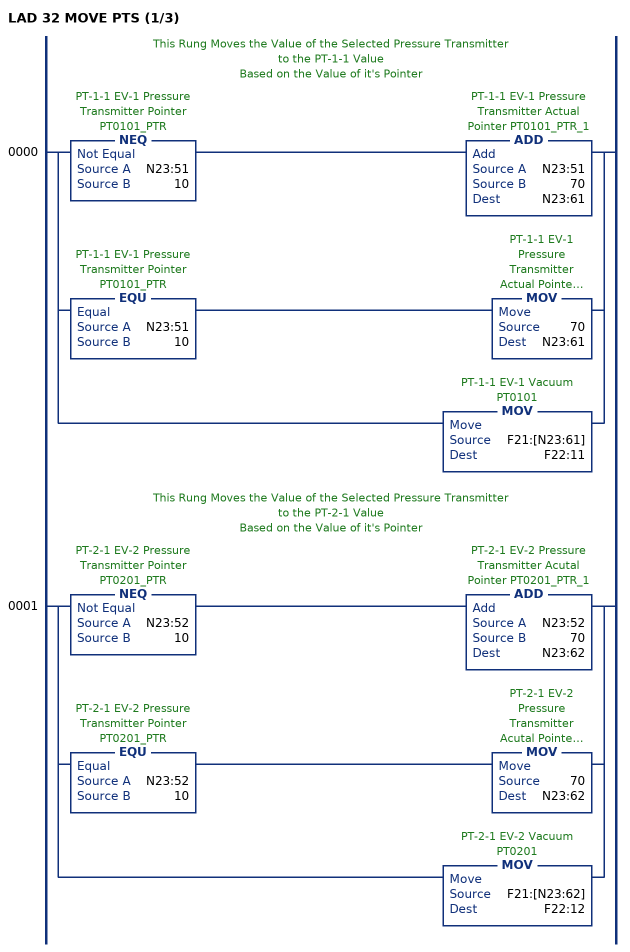
% Rung: 0 %
% This Rung Moves the Value of the Selected Pressure Transmitter
% to the PT-1-1 Value
% Based on the Value of it's Pointer %
SOR BST NEQ N23:51 10 ADD N23:51 70 N23:61 NXB EQU N23:51 10 MOV 70 N23:61 NXB MOV F21:[N23:61] F22:11 BND EOR
%   N23:51  PT0101_PTR  "PT-1-1 EV-1 Pressure Transmitter Pointer" %
%   N23:61  PT0101_PTR_1  "PT-1-1 EV-1 Pressure Transmitter Actual Pointer" %
%   F22:11  PT0101  "PT-1-1 EV-1 Vacuum" %
% Rung: 1 %
% This Rung Moves the Value of the Selected Pressure Transmitter
% to the PT-2-1 Value
% Based on the Value of it's Pointer %
SOR BST NEQ N23:52 10 ADD N23:52 70 N23:62 NXB EQU N23:52 10 MOV 70 N23:62 NXB MOV F21:[N23:62] F22:12 BND EOR
%   N23:52  PT0201_PTR  "PT-2-1 EV-2 Pressure Transmitter Pointer" %
%   N23:62  PT0201_PTR_1  "PT-2-1 EV-2 Pressure Transmitter Acutal Pointer" %
%   F22:12  PT0201  "PT-2-1 EV-2 Vacuum" %

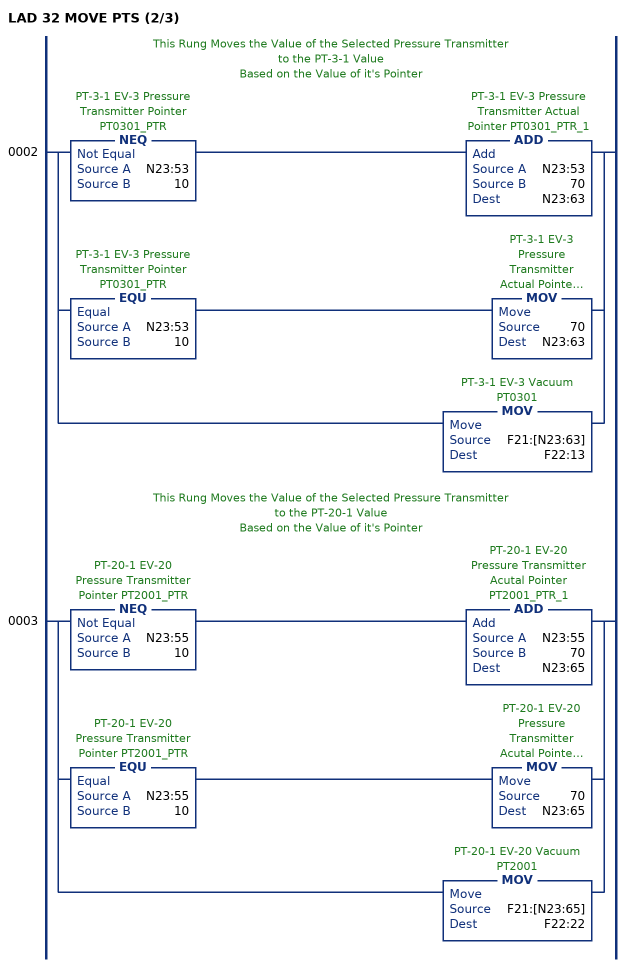
% Rung: 2 %
% This Rung Moves the Value of the Selected Pressure Transmitter
% to the PT-3-1 Value
% Based on the Value of it's Pointer %
SOR BST NEQ N23:53 10 ADD N23:53 70 N23:63 NXB EQU N23:53 10 MOV 70 N23:63 NXB MOV F21:[N23:63] F22:13 BND EOR
%   N23:53  PT0301_PTR  "PT-3-1 EV-3 Pressure Transmitter Pointer" %
%   N23:63  PT0301_PTR_1  "PT-3-1 EV-3 Pressure Transmitter Actual Pointer" %
%   F22:13  PT0301  "PT-3-1 EV-3 Vacuum" %
% Rung: 3 %
% This Rung Moves the Value of the Selected Pressure Transmitter
% to the PT-20-1 Value
% Based on the Value of it's Pointer %
SOR BST NEQ N23:55 10 ADD N23:55 70 N23:65 NXB EQU N23:55 10 MOV 70 N23:65 NXB MOV F21:[N23:65] F22:22 BND EOR
%   N23:55  PT2001_PTR  "PT-20-1 EV-20 Pressure Transmitter Pointer" %
%   N23:65  PT2001_PTR_1  "PT-20-1 EV-20 Pressure Transmitter Acutal Pointer" %
%   F22:22  PT2001  "PT-20-1 EV-20 Vacuum" %

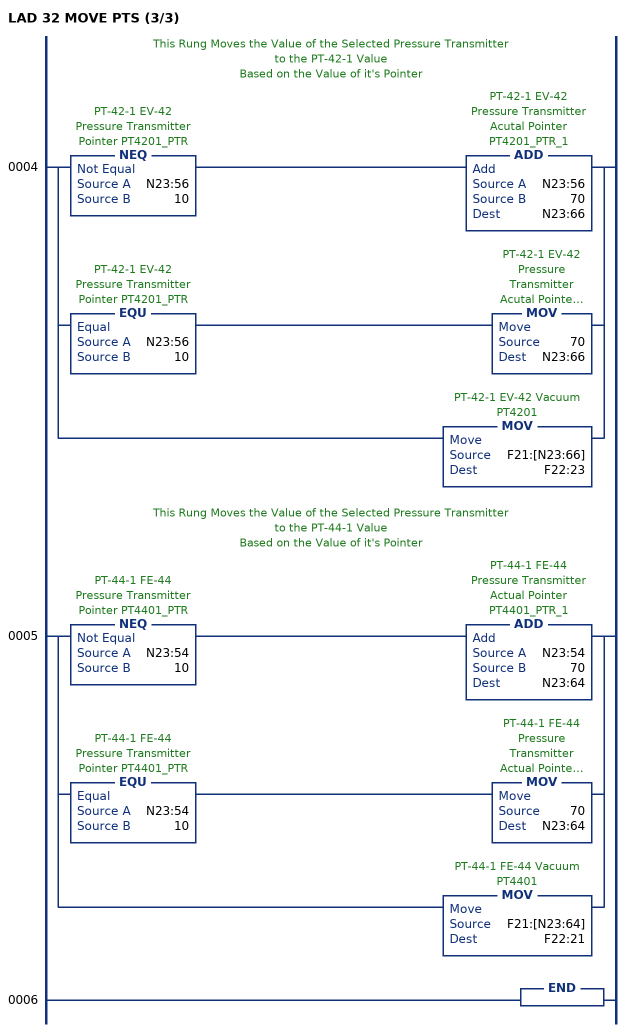
% Rung: 4 %
% This Rung Moves the Value of the Selected Pressure Transmitter
% to the PT-42-1 Value
% Based on the Value of it's Pointer %
SOR BST NEQ N23:56 10 ADD N23:56 70 N23:66 NXB EQU N23:56 10 MOV 70 N23:66 NXB MOV F21:[N23:66] F22:23 BND EOR
%   N23:56  PT4201_PTR  "PT-42-1 EV-42 Pressure Transmitter Pointer" %
%   N23:66  PT4201_PTR_1  "PT-42-1 EV-42 Pressure Transmitter Acutal Pointer" %
%   F22:23  PT4201  "PT-42-1 EV-42 Vacuum" %
% Rung: 5 %
% This Rung Moves the Value of the Selected Pressure Transmitter
% to the PT-44-1 Value
% Based on the Value of it's Pointer %
SOR BST NEQ N23:54 10 ADD N23:54 70 N23:64 NXB EQU N23:54 10 MOV 70 N23:64 NXB MOV F21:[N23:64] F22:21 BND EOR
%   N23:54  PT4401_PTR  "PT-44-1 FE-44 Pressure Transmitter Pointer" %
%   N23:64  PT4401_PTR_1  "PT-44-1 FE-44 Pressure Transmitter Actual Pointer" %
%   F22:21  PT4401  "PT-44-1 FE-44 Vacuum" %
% Rung: 6 %
SOR END EOR

LADDER 33 "MOVE FTS"    % Move FT Info to Sequencial Locations, etc %
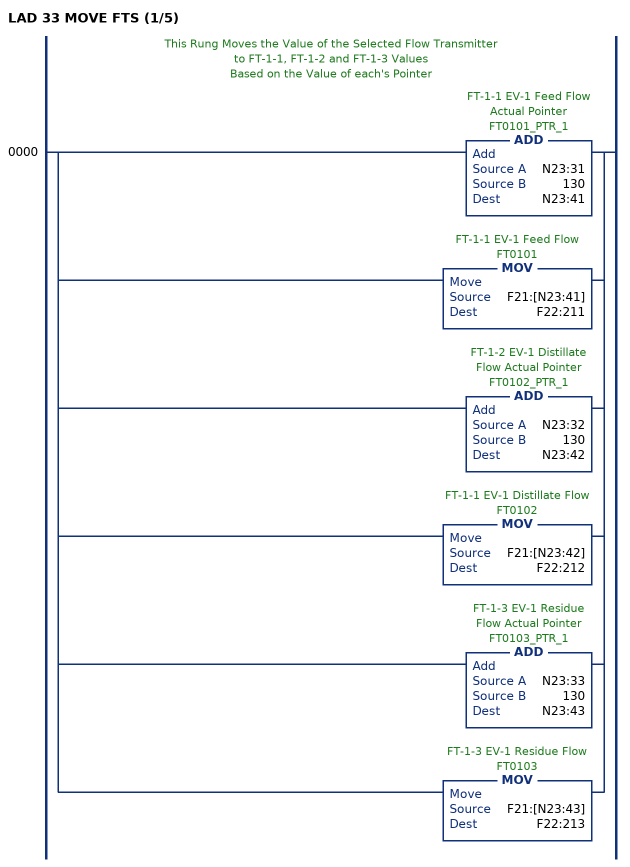
% Rung: 0 %
% This Rung Moves the Value of the Selected Flow Transmitter
% to FT-1-1, FT-1-2 and FT-1-3 Values
% Based on the Value of each's Pointer %
SOR BST ADD N23:31 130 N23:41 NXB MOV F21:[N23:41] F22:211 NXB ADD N23:32 130 N23:42 NXB MOV F21:[N23:42] F22:212 NXB ADD N23:33 130 N23:43 NXB MOV F21:[N23:43] F22:213 BND EOR
%   N23:31  FT0101_PTR  "FT-1-1 EV-1 Feed Flow Pointer" %
%   N23:41  FT0101_PTR_1  "FT-1-1 EV-1 Feed Flow Actual Pointer" %
%   F22:211  FT0101  "FT-1-1 EV-1 Feed Flow" %
%   N23:32  FT0102_PTR  "FT-1-2 EV-1 Distillate Flow Pointer" %
%   N23:42  FT0102_PTR_1  "FT-1-2 EV-1 Distillate Flow Actual Pointer" %
%   F22:212  FT0102  "FT-1-1 EV-1 Distillate Flow" %
%   N23:33  FT0103_PTR  "FT-1-3 EV-1 Residue Flow Pointer" %
%   N23:43  FT0103_PTR_1  "FT-1-3 EV-1 Residue Flow Actual Pointer" %
%   F22:213  FT0103  "FT-1-3 EV-1 Residue Flow" %

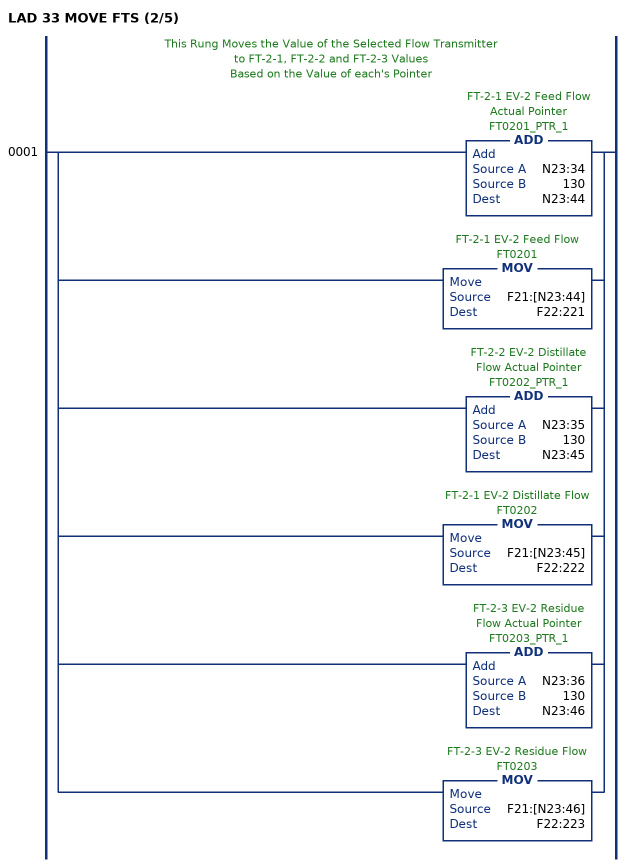
% Rung: 1 %
% This Rung Moves the Value of the Selected Flow Transmitter
% to FT-2-1, FT-2-2 and FT-2-3 Values
% Based on the Value of each's Pointer %
SOR BST ADD N23:34 130 N23:44 NXB MOV F21:[N23:44] F22:221 NXB ADD N23:35 130 N23:45 NXB MOV F21:[N23:45] F22:222 NXB ADD N23:36 130 N23:46 NXB MOV F21:[N23:46] F22:223 BND EOR
%   N23:34  FT0201_PTR  "FT-2-1 EV-2 Feed Flow Pointer" %
%   N23:44  FT0201_PTR_1  "FT-2-1 EV-2 Feed Flow Actual Pointer" %
%   F22:221  FT0201  "FT-2-1 EV-2 Feed Flow" %
%   N23:35  FT0202_PTR  "FT-2-2 EV-2 Distillate Flow Pointer" %
%   N23:45  FT0202_PTR_1  "FT-2-2 EV-2 Distillate Flow Actual Pointer" %
%   F22:222  FT0202  "FT-2-1 EV-2 Distillate Flow" %
%   N23:36  FT0203_PTR  "FT-2-3 EV-2 Residue Flow Pointer" %
%   N23:46  FT0203_PTR_1  "FT-2-3 EV-2 Residue Flow Actual Pointer" %
%   F22:223  FT0203  "FT-2-3 EV-2 Residue Flow" %

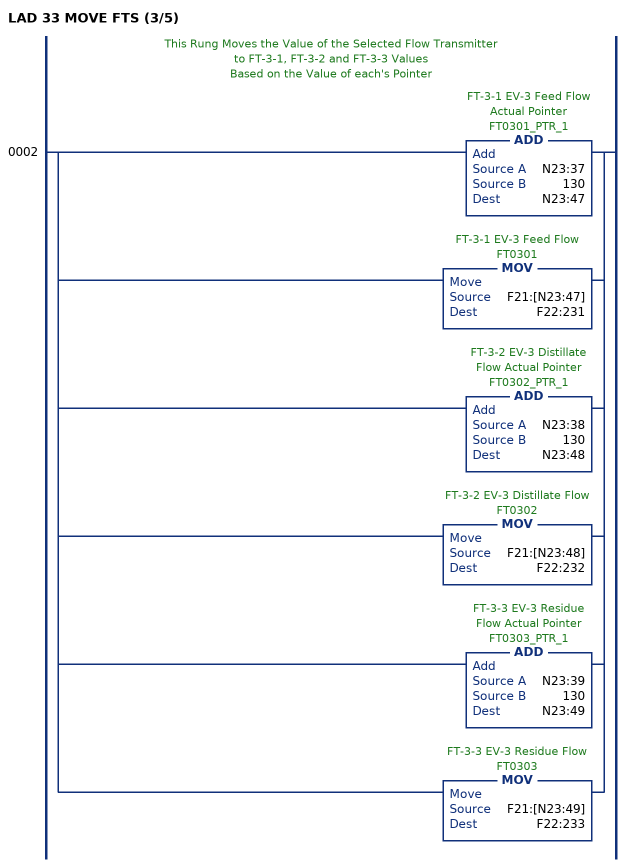
% Rung: 2 %
% This Rung Moves the Value of the Selected Flow Transmitter
% to FT-3-1, FT-3-2 and FT-3-3 Values
% Based on the Value of each's Pointer %
SOR BST ADD N23:37 130 N23:47 NXB MOV F21:[N23:47] F22:231 NXB ADD N23:38 130 N23:48 NXB MOV F21:[N23:48] F22:232 NXB ADD N23:39 130 N23:49 NXB MOV F21:[N23:49] F22:233 BND EOR
%   N23:37  FT0301_PTR  "FT-3-1 EV-3 Feed Flow Pointer" %
%   N23:47  FT0301_PTR_1  "FT-3-1 EV-3 Feed Flow Actual Pointer" %
%   F22:231  FT0301  "FT-3-1 EV-3 Feed Flow" %
%   N23:38  FT0302_PTR  "FT-3-2 EV-3 Distillate Flow Pointer" %
%   N23:48  FT0302_PTR_1  "FT-3-2 EV-3 Distillate Flow Actual Pointer" %
%   F22:232  FT0302  "FT-3-2 EV-3 Distillate Flow" %
%   N23:39  FT0303_PTR  "FT-3-3 EV-3 Residue Flow Pointer" %
%   N23:49  FT0303_PTR_1  "FT-3-3 EV-3 Residue Flow Actual Pointer" %
%   F22:233  FT0303  "FT-3-3 EV-3 Residue Flow" %

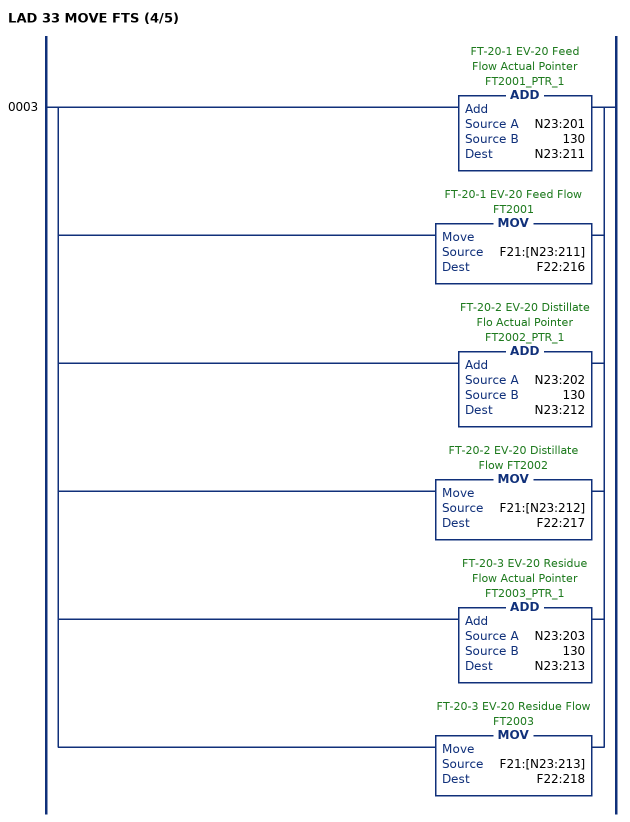
% Rung: 3 %
SOR BST ADD N23:201 130 N23:211 NXB MOV F21:[N23:211] F22:216 NXB ADD N23:202 130 N23:212 NXB MOV F21:[N23:212] F22:217 NXB ADD N23:203 130 N23:213 NXB MOV F21:[N23:213] F22:218 BND EOR
%   N23:201  FT2001_PTR  "FT-20-1 EV-20 Feed Flow Pointer" %
%   N23:211  FT2001_PTR_1  "FT-20-1 EV-20 Feed Flow Actual Pointer" %
%   F22:216  FT2001  "FT-20-1 EV-20 Feed Flow" %
%   N23:202  FT2002_PTR  "FT-20-2 EV-20 Distillate Flo Pointer" %
%   N23:212  FT2002_PTR_1  "FT-20-2 EV-20 Distillate Flo Actual Pointer" %
%   F22:217  FT2002  "FT-20-2 EV-20 Distillate Flow" %
%   N23:203  FT2003_PTR  "FT-20-3 EV-20 Residue Flow Pointer" %
%   N23:213  FT2003_PTR_1  "FT-20-3 EV-20 Residue Flow Actual Pointer" %
%   F22:218  FT2003  "FT-20-3 EV-20 Residue Flow" %

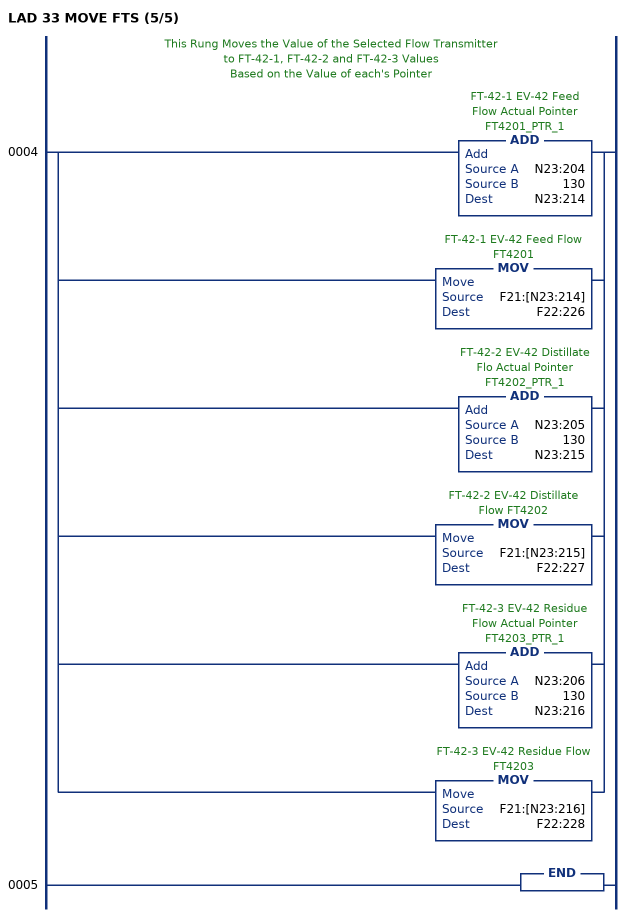
% Rung: 4 %
% This Rung Moves the Value of the Selected Flow Transmitter
% to FT-42-1, FT-42-2 and FT-42-3 Values
% Based on the Value of each's Pointer %
SOR BST ADD N23:204 130 N23:214 NXB MOV F21:[N23:214] F22:226 NXB ADD N23:205 130 N23:215 NXB MOV F21:[N23:215] F22:227 NXB ADD N23:206 130 N23:216 NXB MOV F21:[N23:216] F22:228 BND EOR
%   N23:204  FT4201_PTR  "FT-42-1 EV-42 Feed Flow Pointer" %
%   N23:214  FT4201_PTR_1  "FT-42-1 EV-42 Feed Flow Actual Pointer" %
%   F22:226  FT4201  "FT-42-1 EV-42 Feed Flow" %
%   N23:205  FT4202_PTR  "FT-42-2 EV-42 Distillate Flo Pointer" %
%   N23:215  FT4202_PTR_1  "FT-42-2 EV-42 Distillate Flo Actual Pointer" %
%   F22:227  FT4202  "FT-42-2 EV-42 Distillate Flow" %
%   N23:206  FT4203_PTR  "FT-42-3 EV-42 Residue Flow Pointer" %
%   N23:216  FT4203_PTR_1  "FT-42-3 EV-42 Residue Flow Actual Pointer" %
%   F22:228  FT4203  "FT-42-3 EV-42 Residue Flow" %
% Rung: 5 %
SOR END EOR

LADDER 34 "CALC WTS"    % Convert Remote I/O Data to Real Data for All Scale %
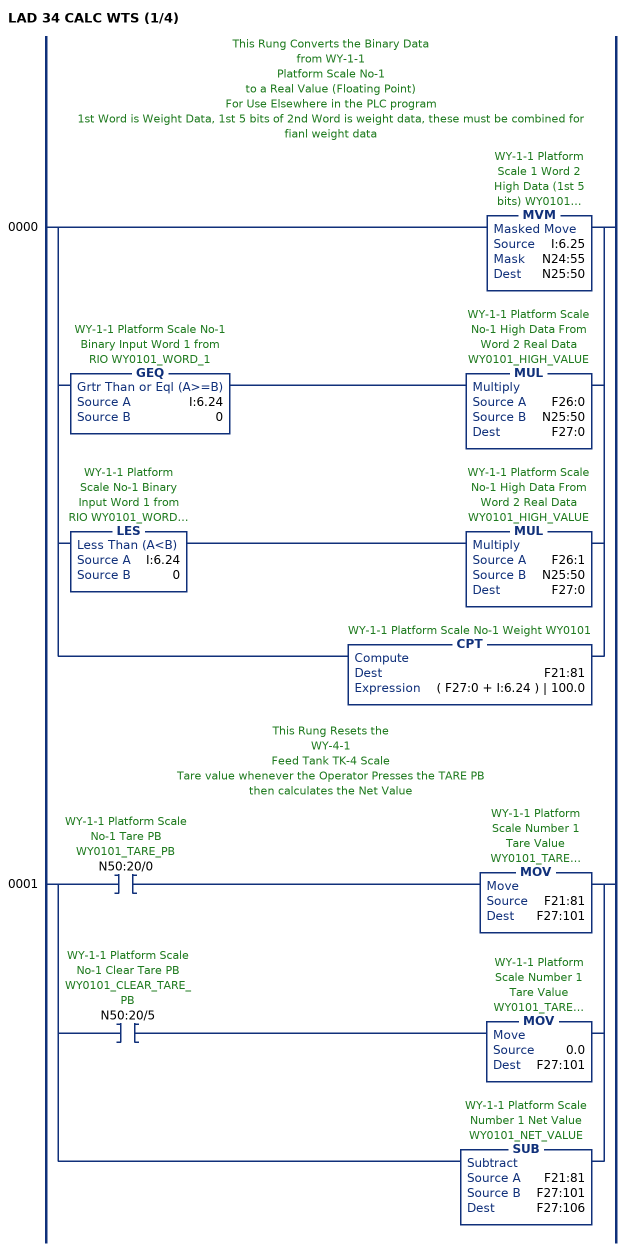
% Rung: 0 %
% This Rung Converts the Binary Data
% from WY-1-1
% Platform Scale No-1
% to a Real Value (Floating Point)
% For Use Elsewhere in the PLC program
% 1st Word is Weight Data, 1st 5 bits of 2nd Word is weight data, these must be combined for fianl weight data %
SOR BST MVM I:6.25 N24:55 N25:50 NXB GEQ I:6.24 0 MUL F26:0 N25:50 F27:0 NXB LES I:6.24 0 MUL F26:1 N25:50 F27:0 NXB CPT F21:81 " ( F27:0 + I:6.24 ) | 100.0 " BND EOR
%   I:6.25  WY0101_WORD_2  "WY-1-1 Platform Scale No-1 Binary Input Word 2 from RIO" %
%   N24:55  WY0101_MASK  "WY-1-1 Platform Scale No-1 Word 2 Mask (Use 1st 5 bits)" %
%   N25:50  WY0101_HIGH_DATA  "WY-1-1 Platform Scale 1 Word 2 High Data (1st 5 bits)" %
%   I:6.24  WY0101_WORD_1  "WY-1-1 Platform Scale No-1 Binary Input Word 1 from RIO" %
%   F26:0  WT_MULTIPLIER_1  "Weigh Scale Multipler if Word 1 >= 0" %
%   F27:0  WY0101_HIGH_VALUE  "WY-1-1 Platform Scale No-1 High Data From Word 2 Real Data" %
%   F26:1  WT_MULTIPLIER_2  "Weigh Scale Multipler if Word 1 < 0" %
%   F21:81  WY0101  "WY-1-1 Platform Scale No-1 Weight" %
% Rung: 1 %
% This Rung Resets the
% WY-4-1
% Feed Tank TK-4 Scale
% Tare value whenever the Operator Presses the TARE PB
% then calculates the Net Value %
SOR BST XIC N50:20/0 MOV F21:81 F27:101 NXB XIC N50:20/5 MOV 0.0 F27:101 NXB SUB F21:81 F27:101 F27:106 BND EOR
%   N50:20/0  WY0101_TARE_PB  "WY-1-1 Platform Scale No-1 Tare PB" %
%   F21:81  WY0101  "WY-1-1 Platform Scale No-1 Weight" %
%   F27:101  WY0101_TARE_VALUE  "WY-1-1 Platform Scale Number 1 Tare Value" %
%   N50:20/5  WY0101_CLEAR_TARE_PB  "WY-1-1 Platform Scale No-1 Clear Tare PB" %
%   F27:106  WY0101_NET_VALUE  "WY-1-1 Platform Scale Number 1 Net Value" %

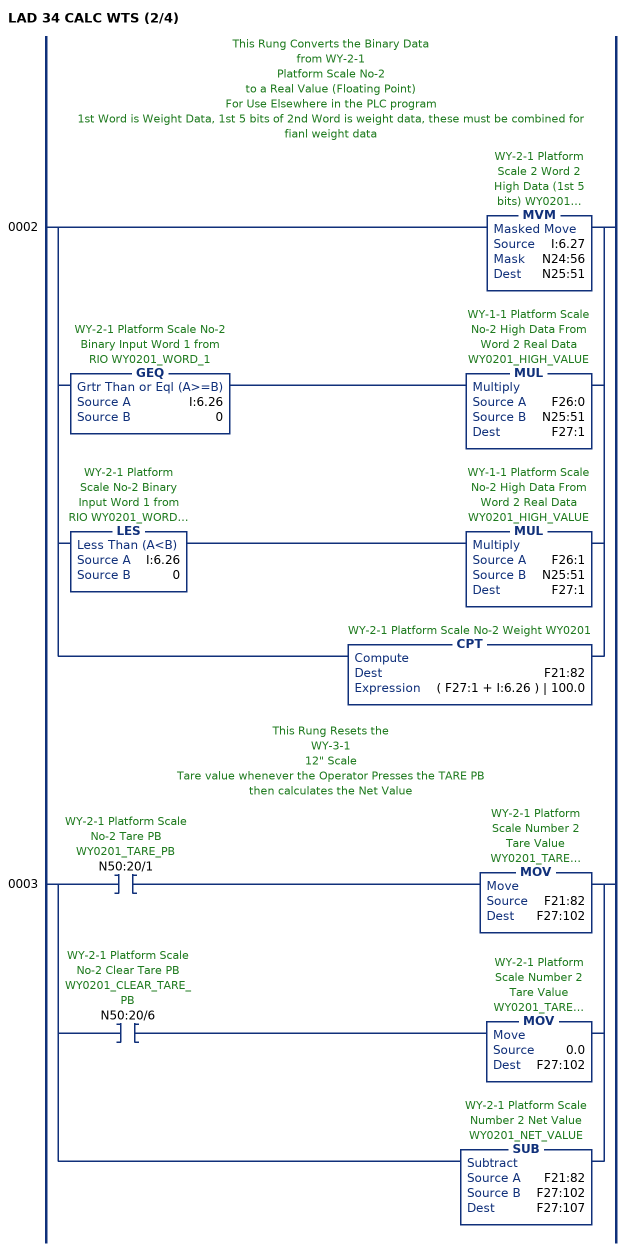
% Rung: 2 %
% This Rung Converts the Binary Data
% from WY-2-1
% Platform Scale No-2
% to a Real Value (Floating Point)
% For Use Elsewhere in the PLC program
% 1st Word is Weight Data, 1st 5 bits of 2nd Word is weight data, these must be combined for fianl weight data %
SOR BST MVM I:6.27 N24:56 N25:51 NXB GEQ I:6.26 0 MUL F26:0 N25:51 F27:1 NXB LES I:6.26 0 MUL F26:1 N25:51 F27:1 NXB CPT F21:82 " ( F27:1 + I:6.26 ) | 100.0 " BND EOR
%   I:6.27  WY0201_WORD_2  "WY-2-1 Platform Scale No-2 Binary Input Word 2 from RIO" %
%   N24:56  WY0201_MASK  "WY-2-1 Platform Scale No-2 Word 2 Mask (Use 1st 5 bits)" %
%   N25:51  WY0201_HIGH_DATA  "WY-2-1 Platform Scale 2 Word 2 High Data (1st 5 bits)" %
%   I:6.26  WY0201_WORD_1  "WY-2-1 Platform Scale No-2 Binary Input Word 1 from RIO" %
%   F26:0  WT_MULTIPLIER_1  "Weigh Scale Multipler if Word 1 >= 0" %
%   F27:1  WY0201_HIGH_VALUE  "WY-1-1 Platform Scale No-2 High Data From Word 2 Real Data" %
%   F26:1  WT_MULTIPLIER_2  "Weigh Scale Multipler if Word 1 < 0" %
%   F21:82  WY0201  "WY-2-1 Platform Scale No-2 Weight" %
% Rung: 3 %
% This Rung Resets the
% WY-3-1
% 12" Scale
% Tare value whenever the Operator Presses the TARE PB
% then calculates the Net Value %
SOR BST XIC N50:20/1 MOV F21:82 F27:102 NXB XIC N50:20/6 MOV 0.0 F27:102 NXB SUB F21:82 F27:102 F27:107 BND EOR
%   N50:20/1  WY0201_TARE_PB  "WY-2-1 Platform Scale No-2 Tare PB" %
%   F21:82  WY0201  "WY-2-1 Platform Scale No-2 Weight" %
%   F27:102  WY0201_TARE_VALUE  "WY-2-1 Platform Scale Number 2 Tare Value" %
%   N50:20/6  WY0201_CLEAR_TARE_PB  "WY-2-1 Platform Scale No-2 Clear Tare PB" %
%   F27:107  WY0201_NET_VALUE  "WY-2-1 Platform Scale Number 2 Net Value" %

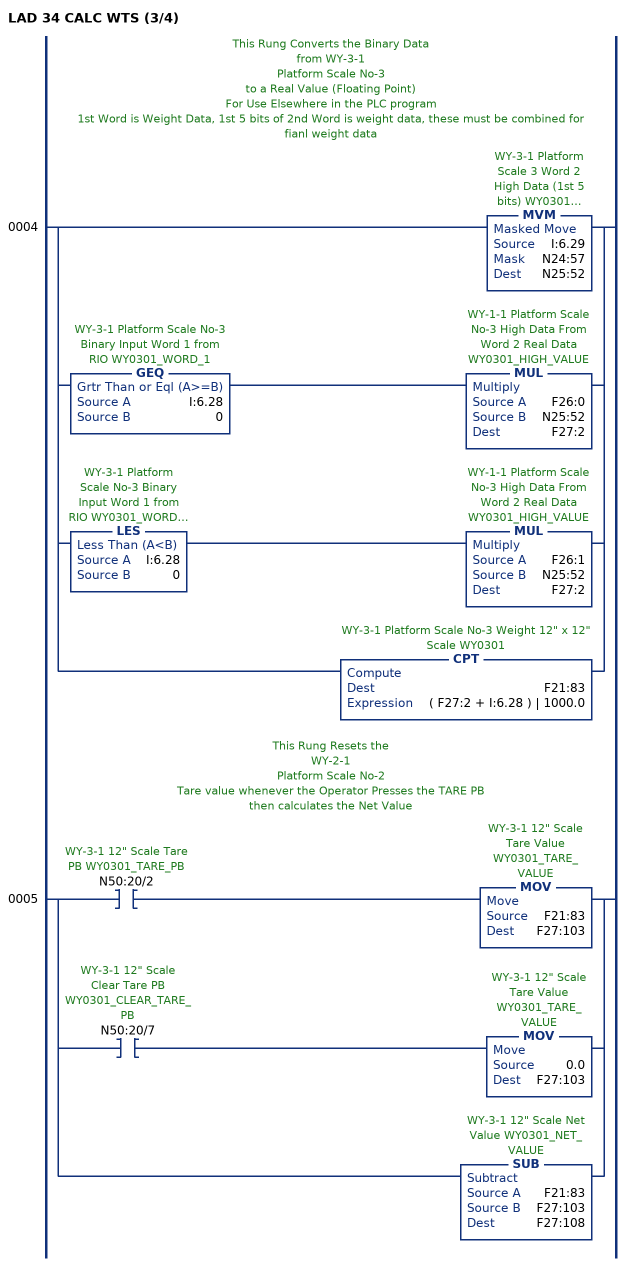
% Rung: 4 %
% This Rung Converts the Binary Data
% from WY-3-1
% Platform Scale No-3
% to a Real Value (Floating Point)
% For Use Elsewhere in the PLC program
% 1st Word is Weight Data, 1st 5 bits of 2nd Word is weight data, these must be combined for fianl weight data %
SOR BST MVM I:6.29 N24:57 N25:52 NXB GEQ I:6.28 0 MUL F26:0 N25:52 F27:2 NXB LES I:6.28 0 MUL F26:1 N25:52 F27:2 NXB CPT F21:83 " ( F27:2 + I:6.28 ) | 1000.0 " BND EOR
%   I:6.29  WY0301_WORD_2  "WY-3-1 Platform Scale No-3 Binary Input Word 2 from RIO" %
%   N24:57  WY0301_MASK  "WY-3-1 Platform Scale No-3 Word 2 Mask (Use 1st 5 bits)" %
%   N25:52  WY0301_HIGH_DATA  "WY-3-1 Platform Scale 3 Word 2 High Data (1st 5 bits)" %
%   I:6.28  WY0301_WORD_1  "WY-3-1 Platform Scale No-3 Binary Input Word 1 from RIO" %
%   F26:0  WT_MULTIPLIER_1  "Weigh Scale Multipler if Word 1 >= 0" %
%   F27:2  WY0301_HIGH_VALUE  "WY-1-1 Platform Scale No-3 High Data From Word 2 Real Data" %
%   F26:1  WT_MULTIPLIER_2  "Weigh Scale Multipler if Word 1 < 0" %
%   F21:83  WY0301  "WY-3-1 Platform Scale No-3 Weight 12" x 12" Scale" %
% Rung: 5 %
% This Rung Resets the
% WY-2-1
% Platform Scale No-2
% Tare value whenever the Operator Presses the TARE PB
% then calculates the Net Value %
SOR BST XIC N50:20/2 MOV F21:83 F27:103 NXB XIC N50:20/7 MOV 0.0 F27:103 NXB SUB F21:83 F27:103 F27:108 BND EOR
%   N50:20/2  WY0301_TARE_PB  "WY-3-1 12" Scale Tare PB" %
%   F21:83  WY0301  "WY-3-1 Platform Scale No-3 Weight 12" x 12" Scale" %
%   F27:103  WY0301_TARE_VALUE  "WY-3-1 12" Scale Tare Value" %
%   N50:20/7  WY0301_CLEAR_TARE_PB  "WY-3-1 12" Scale Clear Tare PB" %
%   F27:108  WY0301_NET_VALUE  "WY-3-1 12" Scale Net Value" %

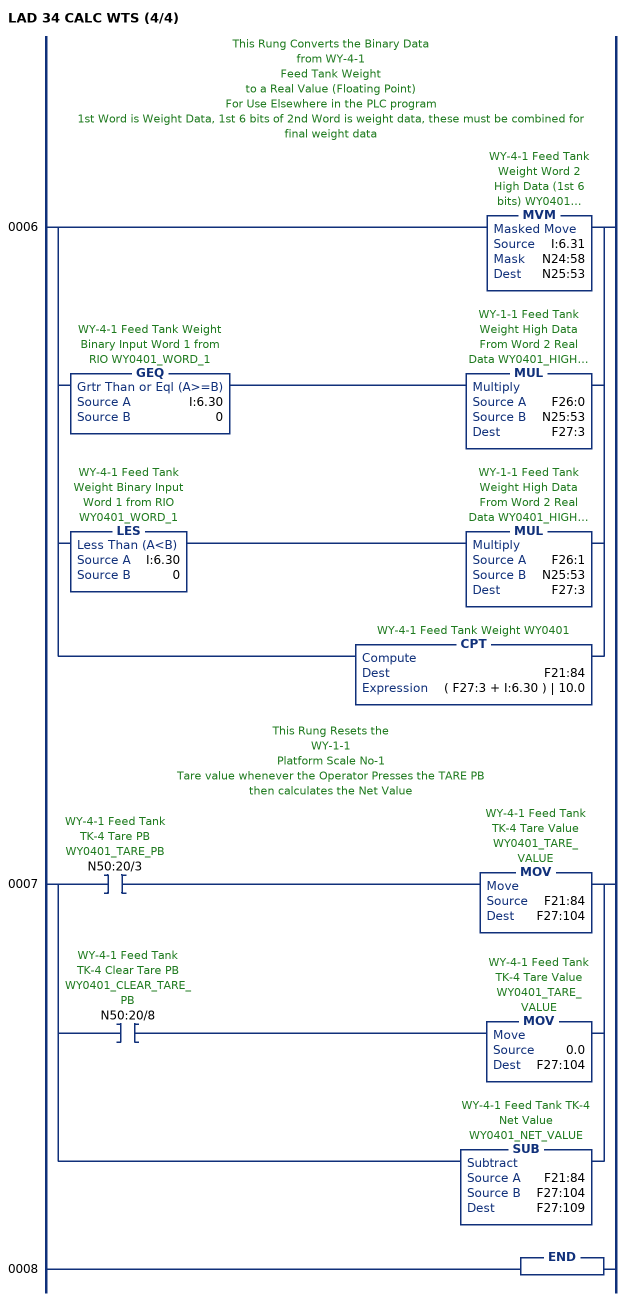
% Rung: 6 %
% This Rung Converts the Binary Data
% from WY-4-1
% Feed Tank Weight
% to a Real Value (Floating Point)
% For Use Elsewhere in the PLC program
% 1st Word is Weight Data, 1st 6 bits of 2nd Word is weight data, these must be combined for final weight data %
SOR BST MVM I:6.31 N24:58 N25:53 NXB GEQ I:6.30 0 MUL F26:0 N25:53 F27:3 NXB LES I:6.30 0 MUL F26:1 N25:53 F27:3 NXB CPT F21:84 " ( F27:3 + I:6.30 ) | 10.0 " BND EOR
%   I:6.31  WY0401_WORD_2  "WY-4-1 Feed Tank Weight Binary Input Word 2 from RIO" %
%   N24:58  WY0401_MASK  "WY-4-1 Feed Tank Weight Word 2 Mask (Use 1st 6 bits)" %
%   N25:53  WY0401_HIGH_DATA  "WY-4-1 Feed Tank Weight Word 2 High Data (1st 6 bits)" %
%   I:6.30  WY0401_WORD_1  "WY-4-1 Feed Tank Weight Binary Input Word 1 from RIO" %
%   F26:0  WT_MULTIPLIER_1  "Weigh Scale Multipler if Word 1 >= 0" %
%   F27:3  WY0401_HIGH_VALUE  "WY-1-1 Feed Tank Weight High Data From Word 2 Real Data" %
%   F26:1  WT_MULTIPLIER_2  "Weigh Scale Multipler if Word 1 < 0" %
%   F21:84  WY0401  "WY-4-1 Feed Tank Weight" %
% Rung: 7 %
% This Rung Resets the
% WY-1-1
% Platform Scale No-1
% Tare value whenever the Operator Presses the TARE PB
% then calculates the Net Value %
SOR BST XIC N50:20/3 MOV F21:84 F27:104 NXB XIC N50:20/8 MOV 0.0 F27:104 NXB SUB F21:84 F27:104 F27:109 BND EOR
%   N50:20/3  WY0401_TARE_PB  "WY-4-1 Feed Tank TK-4 Tare PB" %
%   F21:84  WY0401  "WY-4-1 Feed Tank Weight" %
%   F27:104  WY0401_TARE_VALUE  "WY-4-1 Feed Tank TK-4 Tare Value" %
%   N50:20/8  WY0401_CLEAR_TARE_PB  "WY-4-1 Feed Tank TK-4 Clear Tare PB" %
%   F27:109  WY0401_NET_VALUE  "WY-4-1 Feed Tank TK-4 Net Value" %
% Rung: 8 %
SOR END EOR

LADDER 35 "CALC WT FT"    % Calcualte Flow Rates based on Weight Changes %
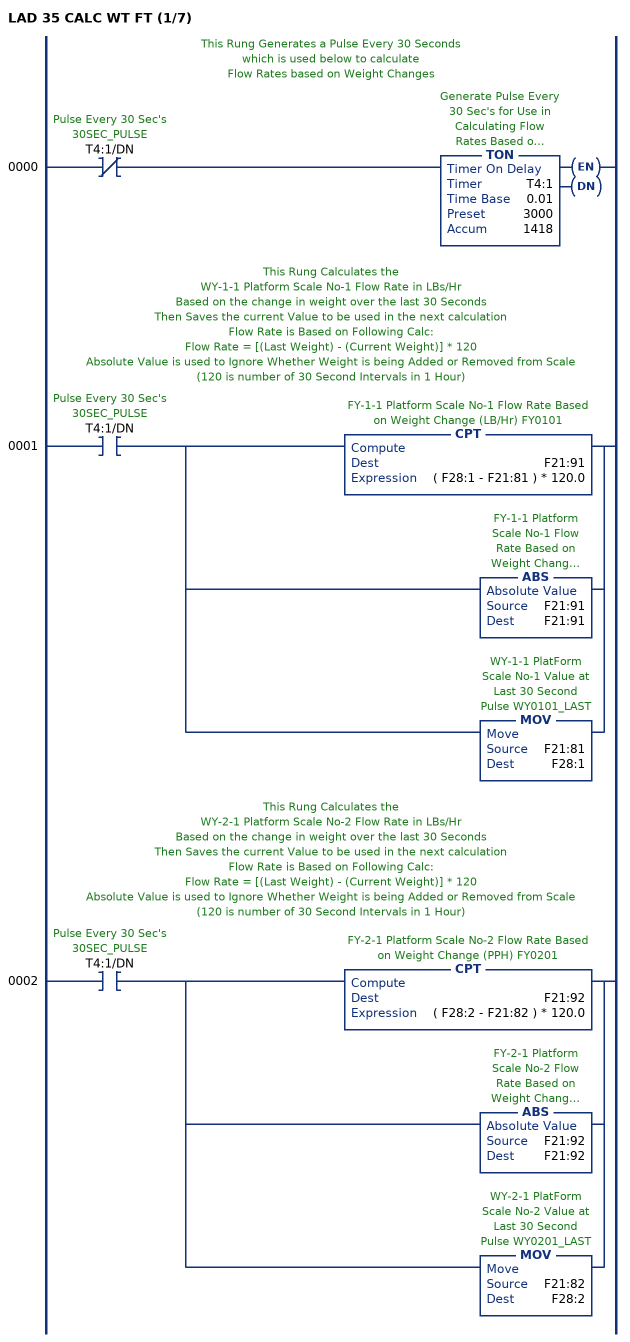
% Rung: 0 %
% This Rung Generates a Pulse Every 30 Seconds
% which is used below to calculate
% Flow Rates based on Weight Changes %
SOR XIO T4:1/DN TON T4:1 0.01 3000 1418 EOR
%   T4:1/DN  30SEC_PULSE  "Pulse Every 30 Sec's" %
%   T4:1  30SEC_TIMER  "Generate Pulse Every 30 Sec's for Use in Calculating Flow Rates Based on Weigh" %
% Rung: 1 %
% This Rung Calculates the
% WY-1-1 Platform Scale No-1 Flow Rate in LBs/Hr
% Based on the change in weight over the last 30 Seconds
% Then Saves the current Value to be used in the next calculation
% Flow Rate is Based on Following Calc:
% 
% Flow Rate = [(Last Weight) - (Current Weight)] * 120
% 
% Absolute Value is used to Ignore Whether Weight is being Added or Removed from Scale
% (120 is number of 30 Second Intervals in 1 Hour) %
SOR XIC T4:1/DN BST CPT F21:91 " ( F28:1 - F21:81 ) * 120.0 " NXB ABS F21:91 F21:91 NXB MOV F21:81 F28:1 BND EOR
%   T4:1/DN  30SEC_PULSE  "Pulse Every 30 Sec's" %
%   F21:91  FY0101  "FY-1-1 Platform Scale No-1 Flow Rate Based on Weight Change (LB/Hr)" %
%   F28:1  WY0101_LAST  "WY-1-1 PlatForm Scale No-1 Value at Last 30 Second Pulse" %
%   F21:81  WY0101  "WY-1-1 Platform Scale No-1 Weight" %
% Rung: 2 %
% This Rung Calculates the
% WY-2-1 Platform Scale No-2 Flow Rate in LBs/Hr
% Based on the change in weight over the last 30 Seconds
% Then Saves the current Value to be used in the next calculation
% Flow Rate is Based on Following Calc:
% 
% Flow Rate = [(Last Weight) - (Current Weight)] * 120
% 
% Absolute Value is used to Ignore Whether Weight is being Added or Removed from Scale
% (120 is number of 30 Second Intervals in 1 Hour) %
SOR XIC T4:1/DN BST CPT F21:92 " ( F28:2 - F21:82 ) * 120.0 " NXB ABS F21:92 F21:92 NXB MOV F21:82 F28:2 BND EOR
%   T4:1/DN  30SEC_PULSE  "Pulse Every 30 Sec's" %
%   F21:92  FY0201  "FY-2-1 Platform Scale No-2 Flow Rate Based on Weight Change (PPH)" %
%   F28:2  WY0201_LAST  "WY-2-1 PlatForm Scale No-2 Value at Last 30 Second Pulse" %
%   F21:82  WY0201  "WY-2-1 Platform Scale No-2 Weight" %

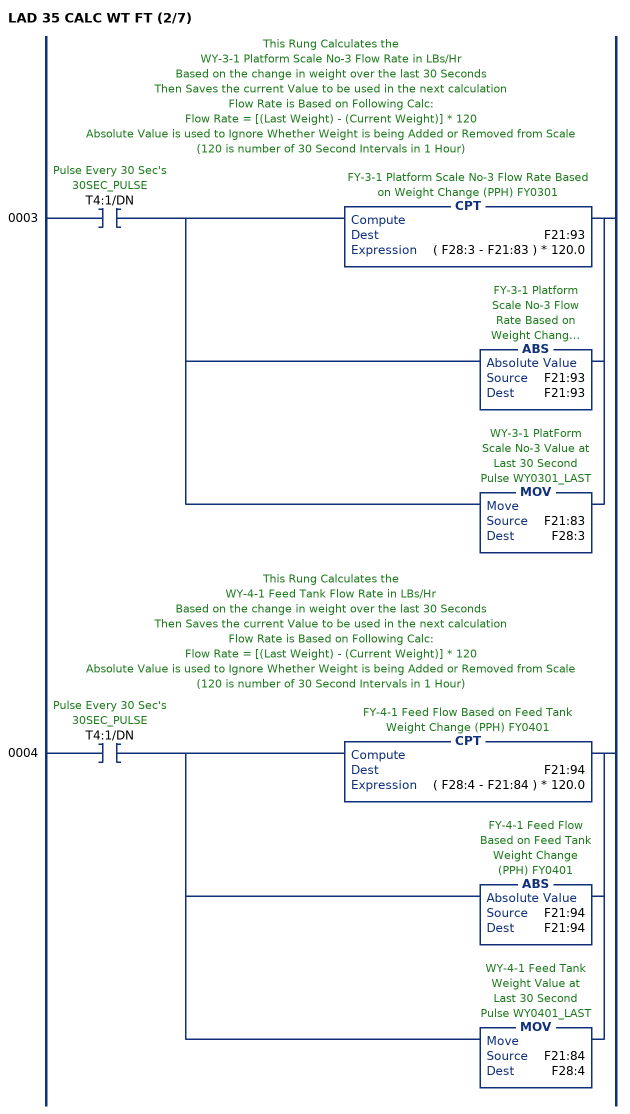
% Rung: 3 %
% This Rung Calculates the
% WY-3-1 Platform Scale No-3 Flow Rate in LBs/Hr
% Based on the change in weight over the last 30 Seconds
% Then Saves the current Value to be used in the next calculation
% Flow Rate is Based on Following Calc:
% 
% Flow Rate = [(Last Weight) - (Current Weight)] * 120
% 
% Absolute Value is used to Ignore Whether Weight is being Added or Removed from Scale
% (120 is number of 30 Second Intervals in 1 Hour) %
SOR XIC T4:1/DN BST CPT F21:93 " ( F28:3 - F21:83 ) * 120.0 " NXB ABS F21:93 F21:93 NXB MOV F21:83 F28:3 BND EOR
%   T4:1/DN  30SEC_PULSE  "Pulse Every 30 Sec's" %
%   F21:93  FY0301  "FY-3-1 Platform Scale No-3 Flow Rate Based on Weight Change (PPH)" %
%   F28:3  WY0301_LAST  "WY-3-1 PlatForm Scale No-3 Value at Last 30 Second Pulse" %
%   F21:83  WY0301  "WY-3-1 Platform Scale No-3 Weight 12" x 12" Scale" %
% Rung: 4 %
% This Rung Calculates the
% WY-4-1 Feed Tank Flow Rate in LBs/Hr
% Based on the change in weight over the last 30 Seconds
% Then Saves the current Value to be used in the next calculation
% Flow Rate is Based on Following Calc:
% 
% Flow Rate = [(Last Weight) - (Current Weight)] * 120
% 
% Absolute Value is used to Ignore Whether Weight is being Added or Removed from Scale
% (120 is number of 30 Second Intervals in 1 Hour) %
SOR XIC T4:1/DN BST CPT F21:94 " ( F28:4 - F21:84 ) * 120.0 " NXB ABS F21:94 F21:94 NXB MOV F21:84 F28:4 BND EOR
%   T4:1/DN  30SEC_PULSE  "Pulse Every 30 Sec's" %
%   F21:94  FY0401  "FY-4-1 Feed Flow Based on Feed Tank Weight Change (PPH)" %
%   F28:4  WY0401_LAST  "WY-4-1 Feed Tank Weight Value at Last 30 Second Pulse" %
%   F21:84  WY0401  "WY-4-1 Feed Tank Weight" %

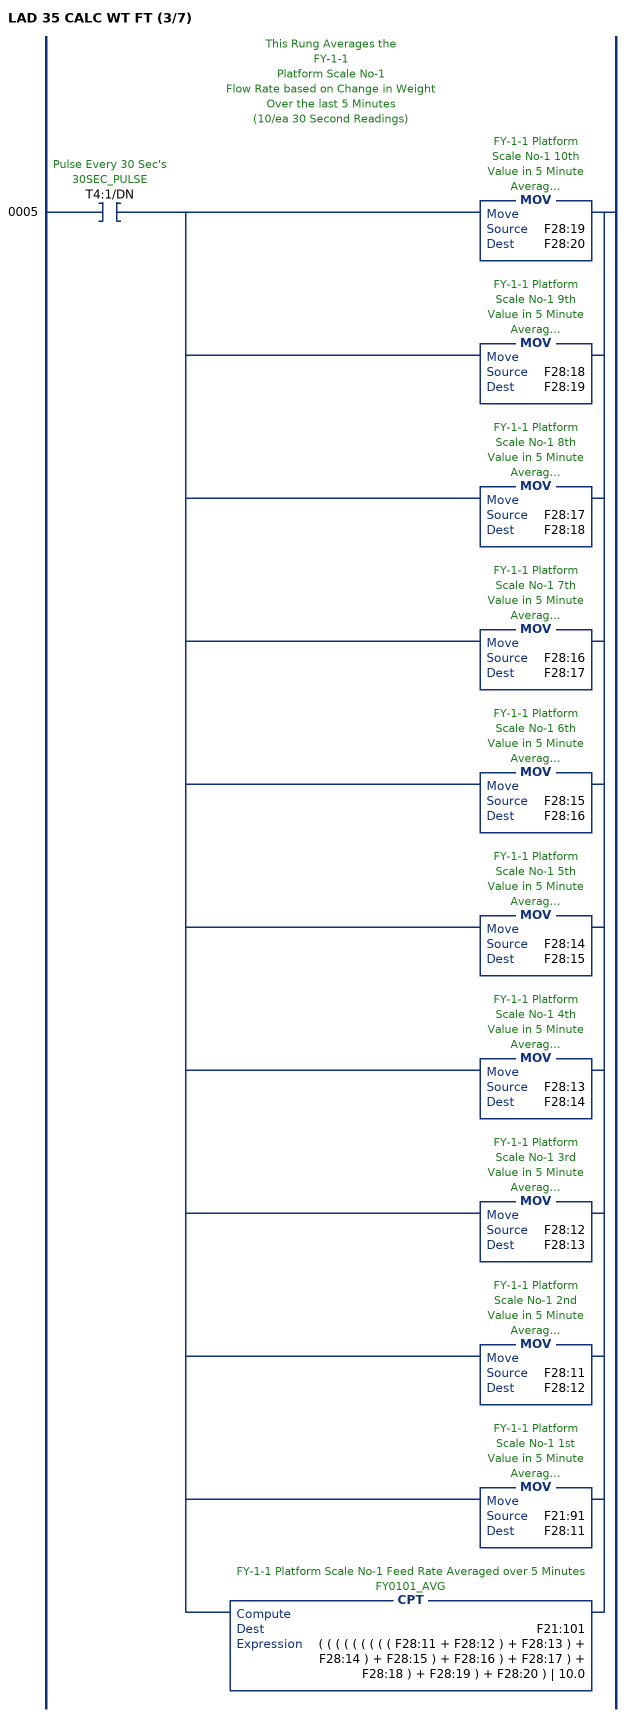
% Rung: 5 %
% This Rung Averages the
% FY-1-1
% Platform Scale No-1
% Flow Rate based on Change in Weight
% Over the last 5 Minutes
% (10/ea 30 Second Readings) %
SOR XIC T4:1/DN BST MOV F28:19 F28:20 NXB MOV F28:18 F28:19 NXB MOV F28:17 F28:18 NXB MOV F28:16 F28:17 NXB MOV F28:15 F28:16 NXB MOV F28:14 F28:15 NXB MOV F28:13 F28:14 NXB MOV F28:12 F28:13 NXB MOV F28:11 F28:12 NXB MOV F21:91 F28:11 NXB CPT F21:101 " ( ( ( ( ( ( ( ( ( F28:11 + F28:12 ) + F28:13 ) + F28:14 ) + F28:15 ) + F28:16 ) + F28:17 ) + F28:18 ) + F28:19 ) + F28:20 ) | 10.0 " BND EOR
%   T4:1/DN  30SEC_PULSE  "Pulse Every 30 Sec's" %
%   F28:19  FY0101_LAST09  "FY-1-1 Platform Scale No-1 9th Value in 5 Minute Average" %
%   F28:20  FY0101_LAST10  "FY-1-1 Platform Scale No-1 10th Value in 5 Minute Average" %
%   F28:18  FY0101_LAST08  "FY-1-1 Platform Scale No-1 8th Value in 5 Minute Average" %
%   F28:17  FY0101_LAST07  "FY-1-1 Platform Scale No-1 7th Value in 5 Minute Average" %
%   F28:16  FY0101_LAST06  "FY-1-1 Platform Scale No-1 6th Value in 5 Minute Average" %
%   F28:15  FY0101_LAST05  "FY-1-1 Platform Scale No-1 5th Value in 5 Minute Average" %
%   F28:14  FY0101_LAST04  "FY-1-1 Platform Scale No-1 4th Value in 5 Minute Average" %
%   F28:13  FY0101_LAST03  "FY-1-1 Platform Scale No-1 3rd Value in 5 Minute Average" %
%   F28:12  FY0101_LAST02  "FY-1-1 Platform Scale No-1 2nd Value in 5 Minute Average" %
%   F28:11  FY0101_LAST01  "FY-1-1 Platform Scale No-1 1st Value in 5 Minute Average" %
%   F21:91  FY0101  "FY-1-1 Platform Scale No-1 Flow Rate Based on Weight Change (LB/Hr)" %
%   F21:101  FY0101_AVG  "FY-1-1 Platform Scale No-1 Feed Rate Averaged over 5 Minutes" %

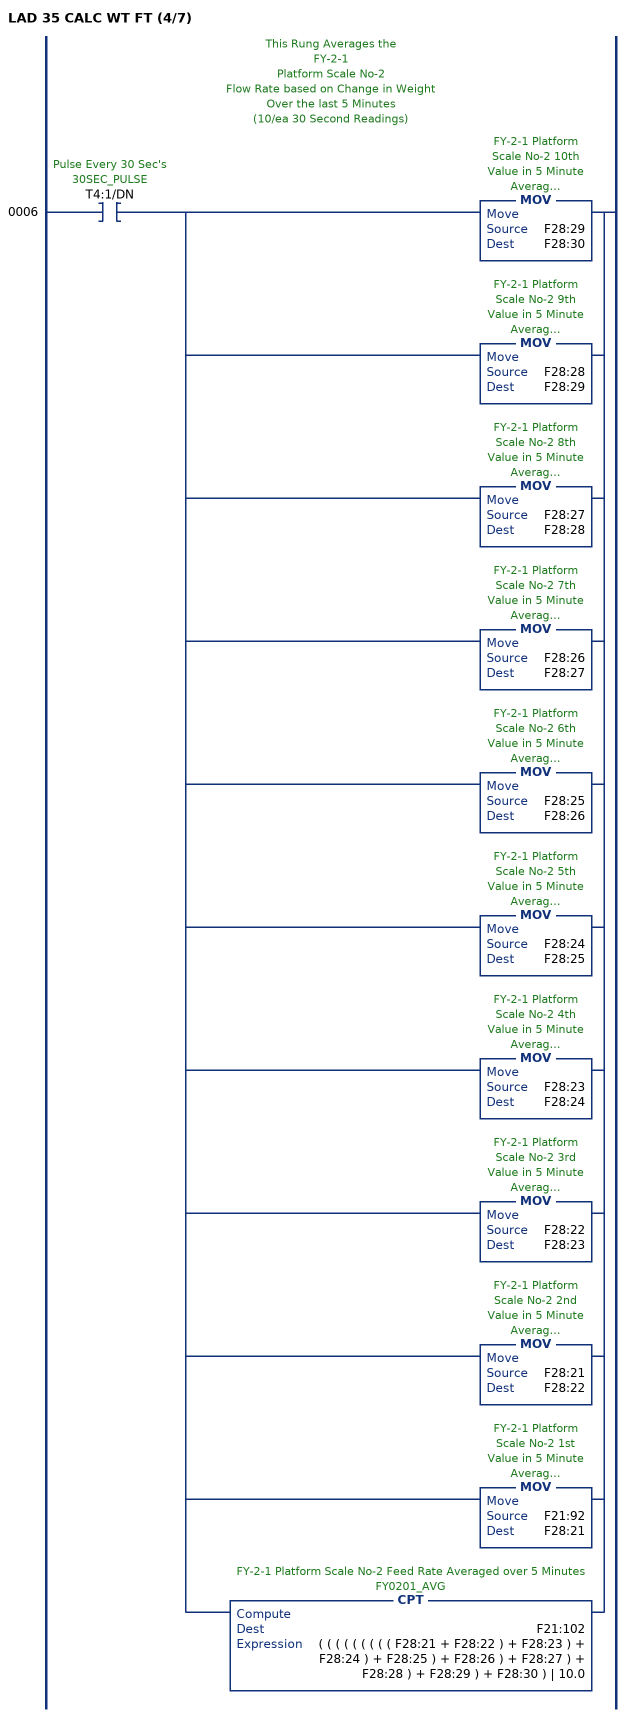
% Rung: 6 %
% This Rung Averages the
% FY-2-1
% Platform Scale No-2
% Flow Rate based on Change in Weight
% Over the last 5 Minutes
% (10/ea 30 Second Readings) %
SOR XIC T4:1/DN BST MOV F28:29 F28:30 NXB MOV F28:28 F28:29 NXB MOV F28:27 F28:28 NXB MOV F28:26 F28:27 NXB MOV F28:25 F28:26 NXB MOV F28:24 F28:25 NXB MOV F28:23 F28:24 NXB MOV F28:22 F28:23 NXB MOV F28:21 F28:22 NXB MOV F21:92 F28:21 NXB CPT F21:102 " ( ( ( ( ( ( ( ( ( F28:21 + F28:22 ) + F28:23 ) + F28:24 ) + F28:25 ) + F28:26 ) + F28:27 ) + F28:28 ) + F28:29 ) + F28:30 ) | 10.0 " BND EOR
%   T4:1/DN  30SEC_PULSE  "Pulse Every 30 Sec's" %
%   F28:29  FY0201_LAST09  "FY-2-1 Platform Scale No-2 9th Value in 5 Minute Average" %
%   F28:30  FY0201_LAST10  "FY-2-1 Platform Scale No-2 10th Value in 5 Minute Average" %
%   F28:28  FY0201_LAST08  "FY-2-1 Platform Scale No-2 8th Value in 5 Minute Average" %
%   F28:27  FY0201_LAST07  "FY-2-1 Platform Scale No-2 7th Value in 5 Minute Average" %
%   F28:26  FY0201_LAST06  "FY-2-1 Platform Scale No-2 6th Value in 5 Minute Average" %
%   F28:25  FY0201_LAST05  "FY-2-1 Platform Scale No-2 5th Value in 5 Minute Average" %
%   F28:24  FY0201_LAST04  "FY-2-1 Platform Scale No-2 4th Value in 5 Minute Average" %
%   F28:23  FY0201_LAST03  "FY-2-1 Platform Scale No-2 3rd Value in 5 Minute Average" %
%   F28:22  FY0201_LAST02  "FY-2-1 Platform Scale No-2 2nd Value in 5 Minute Average" %
%   F28:21  FY0201_LAST01  "FY-2-1 Platform Scale No-2 1st Value in 5 Minute Average" %
%   F21:92  FY0201  "FY-2-1 Platform Scale No-2 Flow Rate Based on Weight Change (PPH)" %
%   F21:102  FY0201_AVG  "FY-2-1 Platform Scale No-2 Feed Rate Averaged over 5 Minutes" %

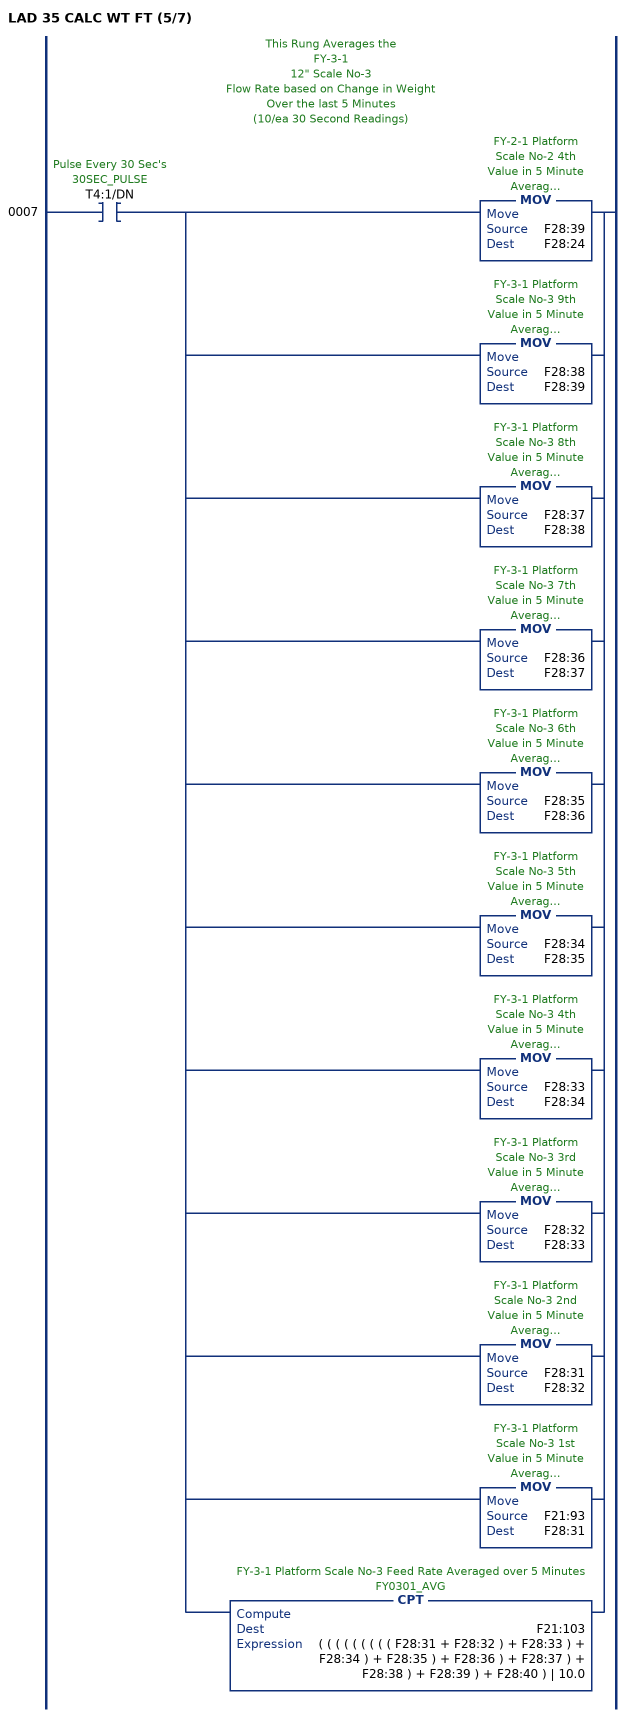
% Rung: 7 %
% This Rung Averages the
% FY-3-1
% 12" Scale No-3
% Flow Rate based on Change in Weight
% Over the last 5 Minutes
% (10/ea 30 Second Readings) %
SOR XIC T4:1/DN BST MOV F28:39 F28:24 NXB MOV F28:38 F28:39 NXB MOV F28:37 F28:38 NXB MOV F28:36 F28:37 NXB MOV F28:35 F28:36 NXB MOV F28:34 F28:35 NXB MOV F28:33 F28:34 NXB MOV F28:32 F28:33 NXB MOV F28:31 F28:32 NXB MOV F21:93 F28:31 NXB CPT F21:103 " ( ( ( ( ( ( ( ( ( F28:31 + F28:32 ) + F28:33 ) + F28:34 ) + F28:35 ) + F28:36 ) + F28:37 ) + F28:38 ) + F28:39 ) + F28:40 ) | 10.0 " BND EOR
%   T4:1/DN  30SEC_PULSE  "Pulse Every 30 Sec's" %
%   F28:39  FY0301_LAST09  "FY-3-1 Platform Scale No-3 9th Value in 5 Minute Average" %
%   F28:24  FY0201_LAST04  "FY-2-1 Platform Scale No-2 4th Value in 5 Minute Average" %
%   F28:38  FY0301_LAST08  "FY-3-1 Platform Scale No-3 8th Value in 5 Minute Average" %
%   F28:37  FY0301_LAST07  "FY-3-1 Platform Scale No-3 7th Value in 5 Minute Average" %
%   F28:36  FY0301_LAST06  "FY-3-1 Platform Scale No-3 6th Value in 5 Minute Average" %
%   F28:35  FY0301_LAST05  "FY-3-1 Platform Scale No-3 5th Value in 5 Minute Average" %
%   F28:34  FY0301_LAST04  "FY-3-1 Platform Scale No-3 4th Value in 5 Minute Average" %
%   F28:33  FY0301_LAST03  "FY-3-1 Platform Scale No-3 3rd Value in 5 Minute Average" %
%   F28:32  FY0301_LAST02  "FY-3-1 Platform Scale No-3 2nd Value in 5 Minute Average" %
%   F28:31  FY0301_LAST01  "FY-3-1 Platform Scale No-3 1st Value in 5 Minute Average" %
%   F21:93  FY0301  "FY-3-1 Platform Scale No-3 Flow Rate Based on Weight Change (PPH)" %
%   F21:103  FY0301_AVG  "FY-3-1 Platform Scale No-3 Feed Rate Averaged over 5 Minutes" %
%   F28:40  FY0301_LAST10  "FY-3-1 Platform Scale No-3 10th Value in 5 Minute Average" %

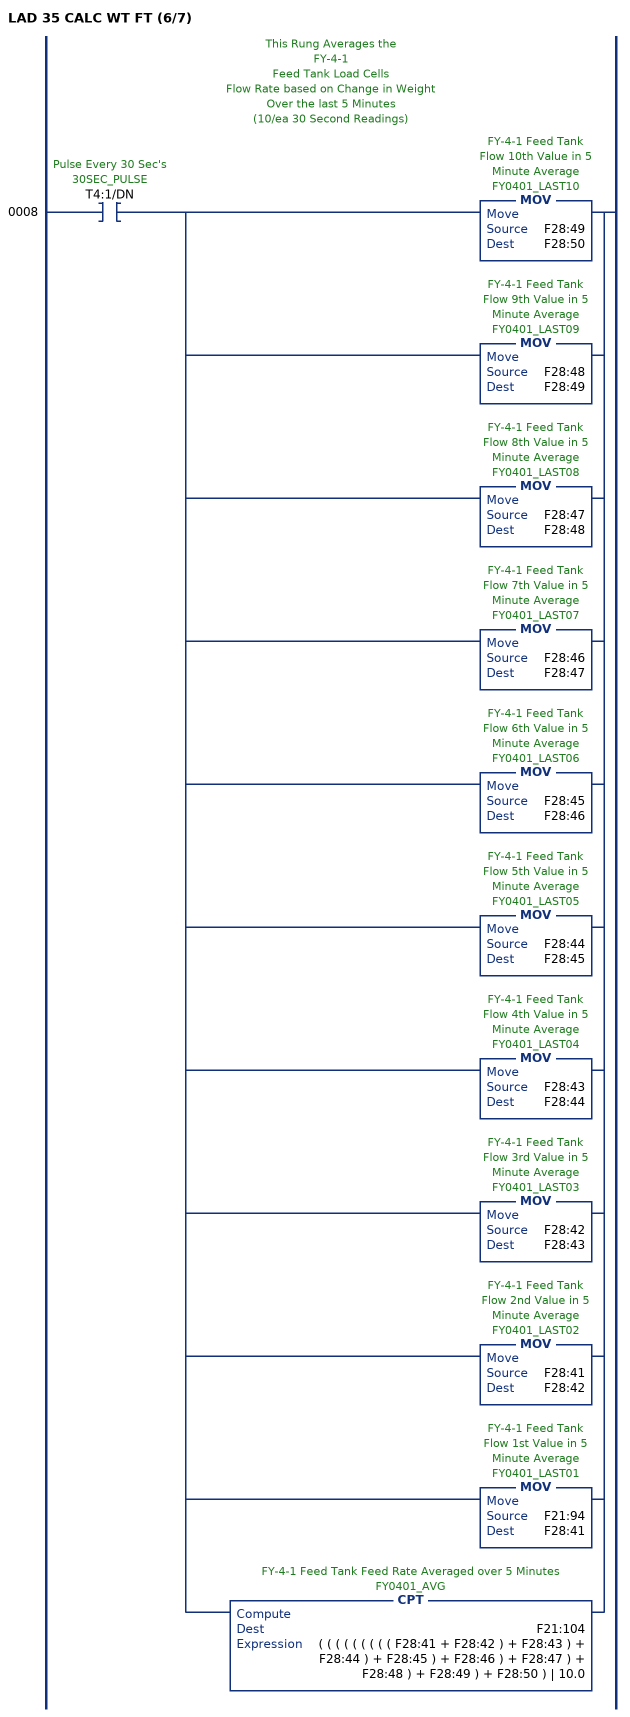
% Rung: 8 %
% This Rung Averages the
% FY-4-1
% Feed Tank Load Cells
% Flow Rate based on Change in Weight
% Over the last 5 Minutes
% (10/ea 30 Second Readings) %
SOR XIC T4:1/DN BST MOV F28:49 F28:50 NXB MOV F28:48 F28:49 NXB MOV F28:47 F28:48 NXB MOV F28:46 F28:47 NXB MOV F28:45 F28:46 NXB MOV F28:44 F28:45 NXB MOV F28:43 F28:44 NXB MOV F28:42 F28:43 NXB MOV F28:41 F28:42 NXB MOV F21:94 F28:41 NXB CPT F21:104 " ( ( ( ( ( ( ( ( ( F28:41 + F28:42 ) + F28:43 ) + F28:44 ) + F28:45 ) + F28:46 ) + F28:47 ) + F28:48 ) + F28:49 ) + F28:50 ) | 10.0 " BND EOR
%   T4:1/DN  30SEC_PULSE  "Pulse Every 30 Sec's" %
%   F28:49  FY0401_LAST09  "FY-4-1 Feed Tank Flow 9th Value in 5 Minute Average" %
%   F28:50  FY0401_LAST10  "FY-4-1 Feed Tank Flow 10th Value in 5 Minute Average" %
%   F28:48  FY0401_LAST08  "FY-4-1 Feed Tank Flow 8th Value in 5 Minute Average" %
%   F28:47  FY0401_LAST07  "FY-4-1 Feed Tank Flow 7th Value in 5 Minute Average" %
%   F28:46  FY0401_LAST06  "FY-4-1 Feed Tank Flow 6th Value in 5 Minute Average" %
%   F28:45  FY0401_LAST05  "FY-4-1 Feed Tank Flow 5th Value in 5 Minute Average" %
%   F28:44  FY0401_LAST04  "FY-4-1 Feed Tank Flow 4th Value in 5 Minute Average" %
%   F28:43  FY0401_LAST03  "FY-4-1 Feed Tank Flow 3rd Value in 5 Minute Average" %
%   F28:42  FY0401_LAST02  "FY-4-1 Feed Tank Flow 2nd Value in 5 Minute Average" %
%   F28:41  FY0401_LAST01  "FY-4-1 Feed Tank Flow 1st Value in 5 Minute Average" %
%   F21:94  FY0401  "FY-4-1 Feed Flow Based on Feed Tank Weight Change (PPH)" %
%   F21:104  FY0401_AVG  "FY-4-1 Feed Tank Feed Rate Averaged over 5 Minutes" %

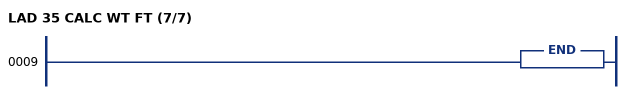
% Rung: 9 %
SOR END EOR

LADDER 36 "CALC PTS"    % Calculate PT's Based on Max & Min Ranges %
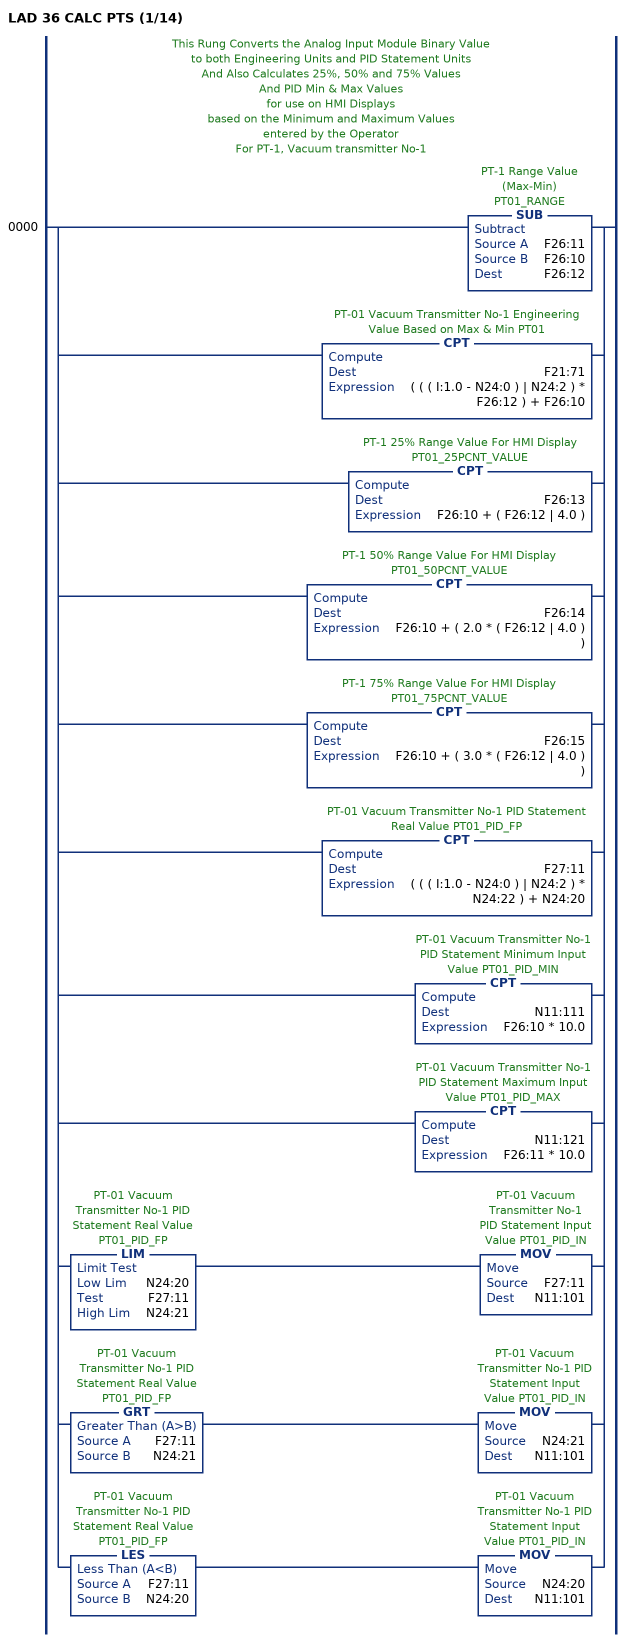
% Rung: 0 %
% This Rung Converts the Analog Input Module Binary Value
% to both Engineering Units and PID Statement Units
% And Also Calculates 25%, 50% and 75% Values
% And PID Min & Max Values
% for use on HMI Displays
% based on the Minimum and Maximum Values
% entered by the Operator
%    For PT-1, Vacuum transmitter No-1 %
SOR BST SUB F26:11 F26:10 F26:12 NXB CPT F21:71 " ( ( ( I:1.0 - N24:0 ) | N24:2 ) * F26:12 ) + F26:10 " NXB CPT F26:13 " F26:10 + ( F26:12 | 4.0 ) " NXB CPT F26:14 " F26:10 + ( 2.0 * ( F26:12 | 4.0 ) ) " NXB CPT F26:15 " F26:10 + ( 3.0 * ( F26:12 | 4.0 ) ) " NXB CPT F27:11 " ( ( ( I:1.0 - N24:0 ) | N24:2 ) * N24:22 ) + N24:20 " NXB CPT N11:111 " F26:10 * 10.0 " NXB CPT N11:121 " F26:11 * 10.0 " NXB LIM N24:20 F27:11 N24:21 MOV F27:11 N11:101 NXB GRT F27:11 N24:21 MOV N24:21 N11:101 NXB LES F27:11 N24:20 MOV N24:20 N11:101 BND EOR
%   F26:11  PT01_MAX  "PT-1 Maximum Value" %
%   F26:10  PT01_MIN  "PT-1 Minimum Value" %
%   F26:12  PT01_RANGE  "PT-1 Range Value (Max-Min)" %
%   F21:71  PT01  "PT-01 Vacuum Transmitter No-1 Engineering Value Based on Max & Min" %
%   I:1.0  PT11_BIN  "PT-1-1 Binary Input From Transmitter Analog Input Module" %
%   N24:0  AI_CURRENT_MIN  "Analog Input Minimum Value = 4 mA DC (From AI Module)" %
%   N24:2  AI_CURRENT_RANGE  "Analog Input Current Range Value = (AI_MAX - AI_MIN) For Use Elswhere" %
%   F26:13  PT01_25PCNT_VALUE  "PT-1 25% Range Value For HMI Display" %
%   F26:14  PT01_50PCNT_VALUE  "PT-1 50% Range Value For HMI Display" %
%   F26:15  PT01_75PCNT_VALUE  "PT-1 75% Range Value For HMI Display" %
%   F27:11  PT01_PID_FP  "PT-01 Vacuum Transmitter No-1 PID Statement Real Value" %
%   N24:22  PID_RANGE  "PID Statement Range Value = (PID_MAX - PID_MIN) For Use Elswhere" %
%   N24:20  PID_MIN  "PID Statement Minimum Value" %
%   N11:111  PT01_PID_MIN  "PT-01 Vacuum Transmitter No-1 PID Statement Minimum Input Value" %
%   N11:121  PT01_PID_MAX  "PT-01 Vacuum Transmitter No-1 PID Statement Maximum Input Value" %
%   N24:21  PID_MAX  "PID Statement Maximum Value" %
%   N11:101  PT01_PID_IN  "PT-01 Vacuum Transmitter No-1 PID Statement Input Value" %

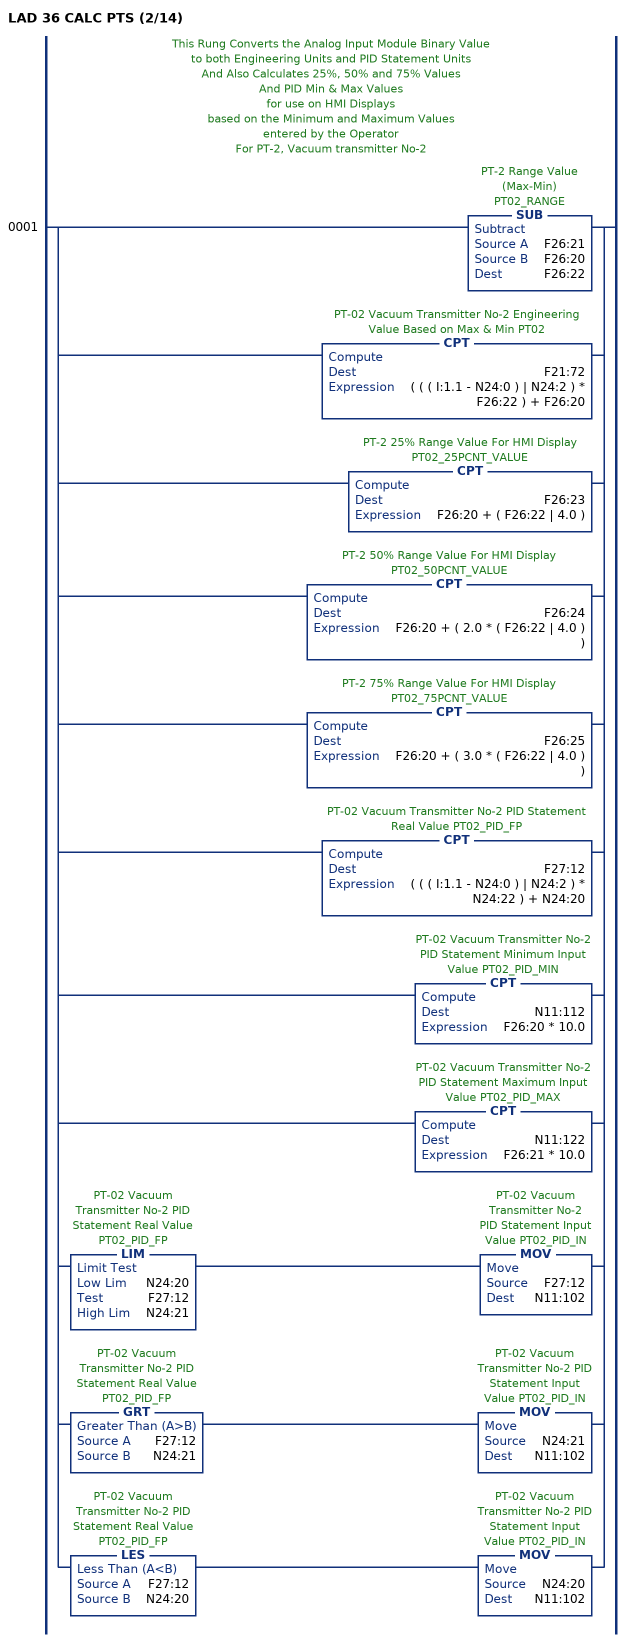
% Rung: 1 %
% This Rung Converts the Analog Input Module Binary Value
% to both Engineering Units and PID Statement Units
% And Also Calculates 25%, 50% and 75% Values
% And PID Min & Max Values
% for use on HMI Displays
% based on the Minimum and Maximum Values
% entered by the Operator
%    For PT-2, Vacuum transmitter No-2 %
SOR BST SUB F26:21 F26:20 F26:22 NXB CPT F21:72 " ( ( ( I:1.1 - N24:0 ) | N24:2 ) * F26:22 ) + F26:20 " NXB CPT F26:23 " F26:20 + ( F26:22 | 4.0 ) " NXB CPT F26:24 " F26:20 + ( 2.0 * ( F26:22 | 4.0 ) ) " NXB CPT F26:25 " F26:20 + ( 3.0 * ( F26:22 | 4.0 ) ) " NXB CPT F27:12 " ( ( ( I:1.1 - N24:0 ) | N24:2 ) * N24:22 ) + N24:20 " NXB CPT N11:112 " F26:20 * 10.0 " NXB CPT N11:122 " F26:21 * 10.0 " NXB LIM N24:20 F27:12 N24:21 MOV F27:12 N11:102 NXB GRT F27:12 N24:21 MOV N24:21 N11:102 NXB LES F27:12 N24:20 MOV N24:20 N11:102 BND EOR
%   F26:21  PT02_MAX  "PT-2 Maximum Value" %
%   F26:20  PT02_MIN  "PT-2 Minimum Value" %
%   F26:22  PT02_RANGE  "PT-2 Range Value (Max-Min)" %
%   F21:72  PT02  "PT-02 Vacuum Transmitter No-2 Engineering Value Based on Max & Min" %
%   I:1.1  PT21_BIN  "PT-2-1 Binary Input From Transmitter Analog Input Module" %
%   N24:0  AI_CURRENT_MIN  "Analog Input Minimum Value = 4 mA DC (From AI Module)" %
%   N24:2  AI_CURRENT_RANGE  "Analog Input Current Range Value = (AI_MAX - AI_MIN) For Use Elswhere" %
%   F26:23  PT02_25PCNT_VALUE  "PT-2 25% Range Value For HMI Display" %
%   F26:24  PT02_50PCNT_VALUE  "PT-2 50% Range Value For HMI Display" %
%   F26:25  PT02_75PCNT_VALUE  "PT-2 75% Range Value For HMI Display" %
%   F27:12  PT02_PID_FP  "PT-02 Vacuum Transmitter No-2 PID Statement Real Value" %
%   N24:22  PID_RANGE  "PID Statement Range Value = (PID_MAX - PID_MIN) For Use Elswhere" %
%   N24:20  PID_MIN  "PID Statement Minimum Value" %
%   N11:112  PT02_PID_MIN  "PT-02 Vacuum Transmitter No-2 PID Statement Minimum Input Value" %
%   N11:122  PT02_PID_MAX  "PT-02 Vacuum Transmitter No-2 PID Statement Maximum Input Value" %
%   N24:21  PID_MAX  "PID Statement Maximum Value" %
%   N11:102  PT02_PID_IN  "PT-02 Vacuum Transmitter No-2 PID Statement Input Value" %

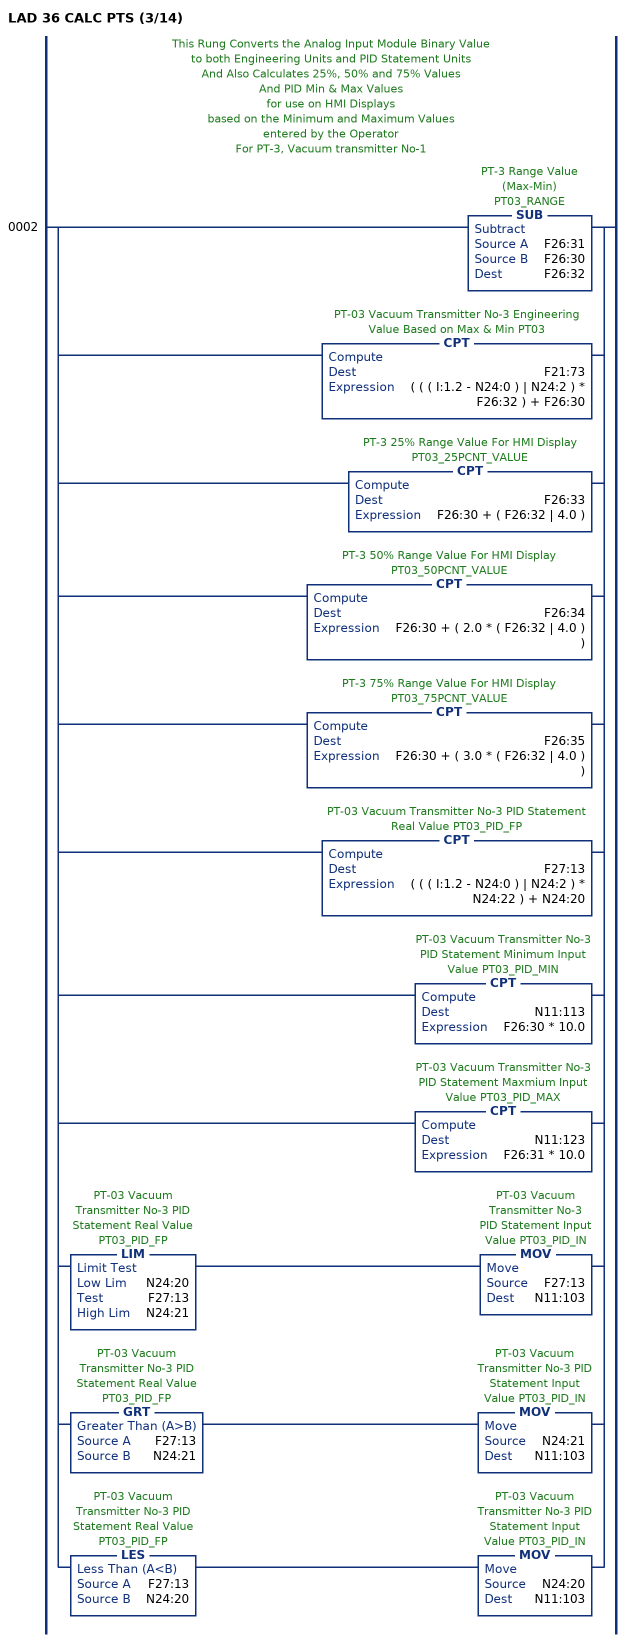
% Rung: 2 %
% This Rung Converts the Analog Input Module Binary Value
% to both Engineering Units and PID Statement Units
% And Also Calculates 25%, 50% and 75% Values
% And PID Min & Max Values
% for use on HMI Displays
% based on the Minimum and Maximum Values
% entered by the Operator
%    For PT-3, Vacuum transmitter No-1 %
SOR BST SUB F26:31 F26:30 F26:32 NXB CPT F21:73 " ( ( ( I:1.2 - N24:0 ) | N24:2 ) * F26:32 ) + F26:30 " NXB CPT F26:33 " F26:30 + ( F26:32 | 4.0 ) " NXB CPT F26:34 " F26:30 + ( 2.0 * ( F26:32 | 4.0 ) ) " NXB CPT F26:35 " F26:30 + ( 3.0 * ( F26:32 | 4.0 ) ) " NXB CPT F27:13 " ( ( ( I:1.2 - N24:0 ) | N24:2 ) * N24:22 ) + N24:20 " NXB CPT N11:113 " F26:30 * 10.0 " NXB CPT N11:123 " F26:31 * 10.0 " NXB LIM N24:20 F27:13 N24:21 MOV F27:13 N11:103 NXB GRT F27:13 N24:21 MOV N24:21 N11:103 NXB LES F27:13 N24:20 MOV N24:20 N11:103 BND EOR
%   F26:31  PT03_MAX  "PT-3 Maximum Value" %
%   F26:30  PT03_MIN  "PT-3 Minimum Value" %
%   F26:32  PT03_RANGE  "PT-3 Range Value (Max-Min)" %
%   F21:73  PT03  "PT-03 Vacuum Transmitter No-3 Engineering Value Based on Max & Min" %
%   I:1.2  PT31_BIN  "PT-3-1 Binary Input From Transmitter Analog Input Module" %
%   N24:0  AI_CURRENT_MIN  "Analog Input Minimum Value = 4 mA DC (From AI Module)" %
%   N24:2  AI_CURRENT_RANGE  "Analog Input Current Range Value = (AI_MAX - AI_MIN) For Use Elswhere" %
%   F26:33  PT03_25PCNT_VALUE  "PT-3 25% Range Value For HMI Display" %
%   F26:34  PT03_50PCNT_VALUE  "PT-3 50% Range Value For HMI Display" %
%   F26:35  PT03_75PCNT_VALUE  "PT-3 75% Range Value For HMI Display" %
%   F27:13  PT03_PID_FP  "PT-03 Vacuum Transmitter No-3 PID Statement Real Value" %
%   N24:22  PID_RANGE  "PID Statement Range Value = (PID_MAX - PID_MIN) For Use Elswhere" %
%   N24:20  PID_MIN  "PID Statement Minimum Value" %
%   N11:113  PT03_PID_MIN  "PT-03 Vacuum Transmitter No-3 PID Statement Minimum Input Value" %
%   N11:123  PT03_PID_MAX  "PT-03 Vacuum Transmitter No-3 PID Statement Maxmium Input Value" %
%   N24:21  PID_MAX  "PID Statement Maximum Value" %
%   N11:103  PT03_PID_IN  "PT-03 Vacuum Transmitter No-3 PID Statement Input Value" %

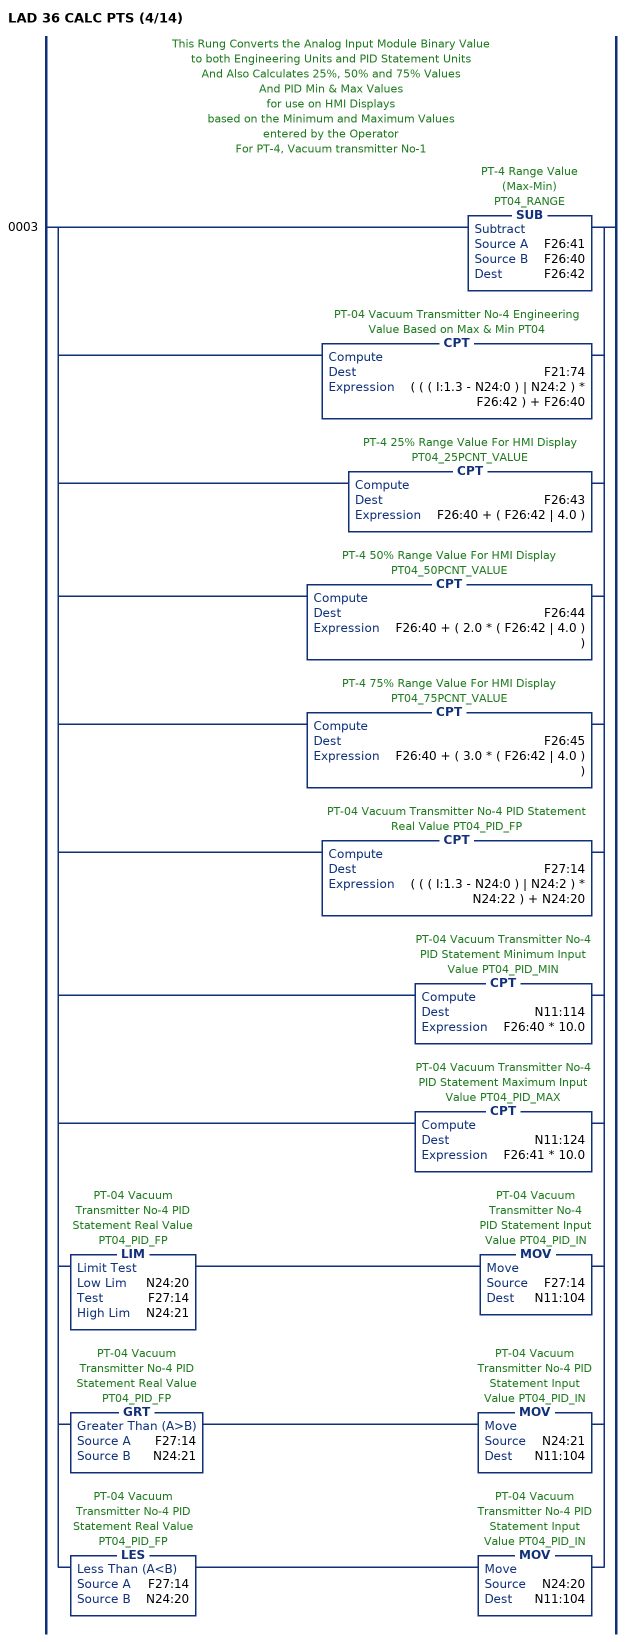
% Rung: 3 %
% This Rung Converts the Analog Input Module Binary Value
% to both Engineering Units and PID Statement Units
% And Also Calculates 25%, 50% and 75% Values
% And PID Min & Max Values
% for use on HMI Displays
% based on the Minimum and Maximum Values
% entered by the Operator
%    For PT-4, Vacuum transmitter No-1 %
SOR BST SUB F26:41 F26:40 F26:42 NXB CPT F21:74 " ( ( ( I:1.3 - N24:0 ) | N24:2 ) * F26:42 ) + F26:40 " NXB CPT F26:43 " F26:40 + ( F26:42 | 4.0 ) " NXB CPT F26:44 " F26:40 + ( 2.0 * ( F26:42 | 4.0 ) ) " NXB CPT F26:45 " F26:40 + ( 3.0 * ( F26:42 | 4.0 ) ) " NXB CPT F27:14 " ( ( ( I:1.3 - N24:0 ) | N24:2 ) * N24:22 ) + N24:20 " NXB CPT N11:114 " F26:40 * 10.0 " NXB CPT N11:124 " F26:41 * 10.0 " NXB LIM N24:20 F27:14 N24:21 MOV F27:14 N11:104 NXB GRT F27:14 N24:21 MOV N24:21 N11:104 NXB LES F27:14 N24:20 MOV N24:20 N11:104 BND EOR
%   F26:41  PT04_MAX  "PT-4 Maximum Value" %
%   F26:40  PT04_MIN  "PT-4 Minimum Value" %
%   F26:42  PT04_RANGE  "PT-4 Range Value (Max-Min)" %
%   F21:74  PT04  "PT-04 Vacuum Transmitter No-4 Engineering Value Based on Max & Min" %
%   I:1.3  PT41_BIN  "PT-4-1 Binary Input From Transmitter Analog Input Module" %
%   N24:0  AI_CURRENT_MIN  "Analog Input Minimum Value = 4 mA DC (From AI Module)" %
%   N24:2  AI_CURRENT_RANGE  "Analog Input Current Range Value = (AI_MAX - AI_MIN) For Use Elswhere" %
%   F26:43  PT04_25PCNT_VALUE  "PT-4 25% Range Value For HMI Display" %
%   F26:44  PT04_50PCNT_VALUE  "PT-4 50% Range Value For HMI Display" %
%   F26:45  PT04_75PCNT_VALUE  "PT-4 75% Range Value For HMI Display" %
%   F27:14  PT04_PID_FP  "PT-04 Vacuum Transmitter No-4 PID Statement Real Value" %
%   N24:22  PID_RANGE  "PID Statement Range Value = (PID_MAX - PID_MIN) For Use Elswhere" %
%   N24:20  PID_MIN  "PID Statement Minimum Value" %
%   N11:114  PT04_PID_MIN  "PT-04 Vacuum Transmitter No-4 PID Statement Minimum Input Value" %
%   N11:124  PT04_PID_MAX  "PT-04 Vacuum Transmitter No-4 PID Statement Maximum Input Value" %
%   N24:21  PID_MAX  "PID Statement Maximum Value" %
%   N11:104  PT04_PID_IN  "PT-04 Vacuum Transmitter No-4 PID Statement Input Value" %

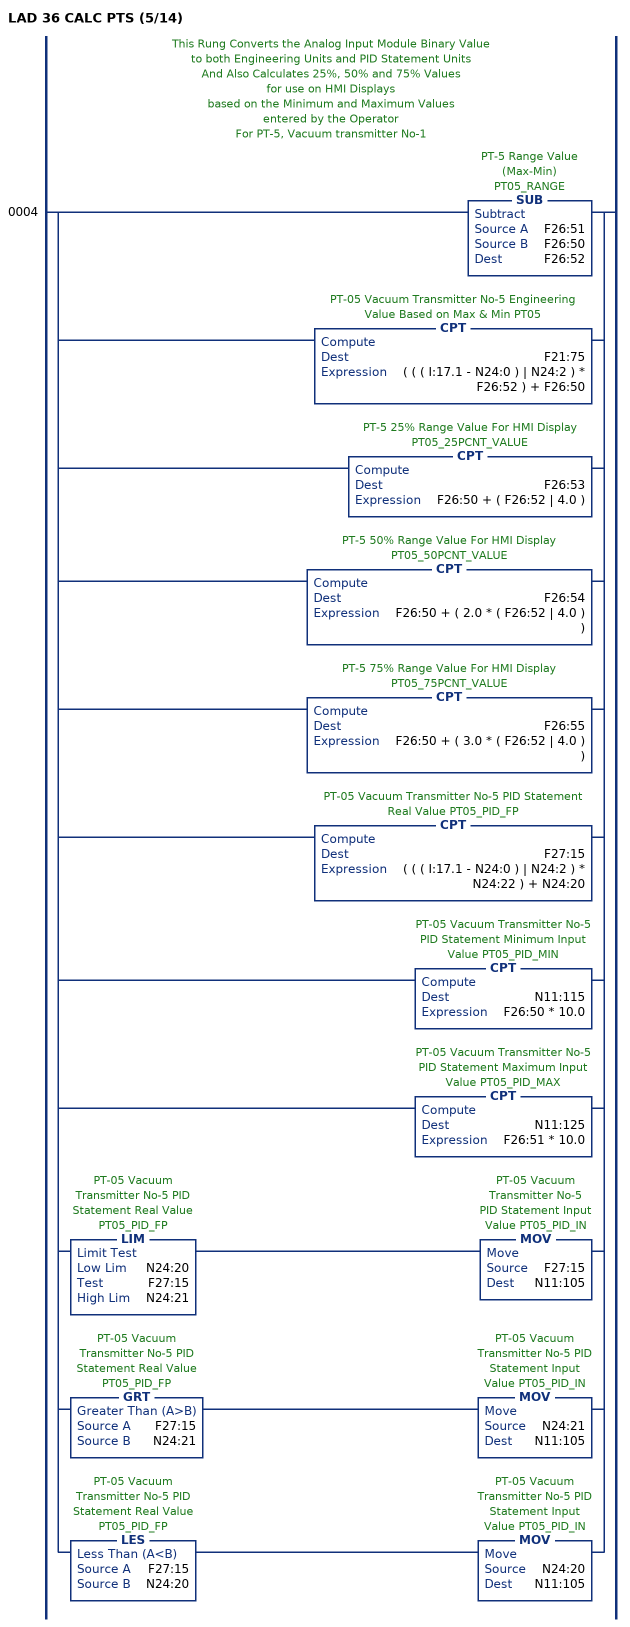
% Rung: 4 %
% This Rung Converts the Analog Input Module Binary Value
% to both Engineering Units and PID Statement Units
% And Also Calculates 25%, 50% and 75% Values
% for use on HMI Displays
% based on the Minimum and Maximum Values
% entered by the Operator
%    For PT-5, Vacuum transmitter No-1 %
SOR BST SUB F26:51 F26:50 F26:52 NXB CPT F21:75 " ( ( ( I:17.1 - N24:0 ) | N24:2 ) * F26:52 ) + F26:50 " NXB CPT F26:53 " F26:50 + ( F26:52 | 4.0 ) " NXB CPT F26:54 " F26:50 + ( 2.0 * ( F26:52 | 4.0 ) ) " NXB CPT F26:55 " F26:50 + ( 3.0 * ( F26:52 | 4.0 ) ) " NXB CPT F27:15 " ( ( ( I:17.1 - N24:0 ) | N24:2 ) * N24:22 ) + N24:20 " NXB CPT N11:115 " F26:50 * 10.0 " NXB CPT N11:125 " F26:51 * 10.0 " NXB LIM N24:20 F27:15 N24:21 MOV F27:15 N11:105 NXB GRT F27:15 N24:21 MOV N24:21 N11:105 NXB LES F27:15 N24:20 MOV N24:20 N11:105 BND EOR
%   F26:51  PT05_MAX  "PT-5 Maximum Value" %
%   F26:50  PT05_MIN  "PT-5 Minimum Value" %
%   F26:52  PT05_RANGE  "PT-5 Range Value (Max-Min)" %
%   F21:75  PT05  "PT-05 Vacuum Transmitter No-5 Engineering Value Based on Max & Min" %
%   I:17.1  PT51_BIN  "PT-5 Binary Input From Transmitter Analog Input Module" %
%   N24:0  AI_CURRENT_MIN  "Analog Input Minimum Value = 4 mA DC (From AI Module)" %
%   N24:2  AI_CURRENT_RANGE  "Analog Input Current Range Value = (AI_MAX - AI_MIN) For Use Elswhere" %
%   F26:53  PT05_25PCNT_VALUE  "PT-5 25% Range Value For HMI Display" %
%   F26:54  PT05_50PCNT_VALUE  "PT-5 50% Range Value For HMI Display" %
%   F26:55  PT05_75PCNT_VALUE  "PT-5 75% Range Value For HMI Display" %
%   F27:15  PT05_PID_FP  "PT-05 Vacuum Transmitter No-5 PID Statement Real Value" %
%   N24:22  PID_RANGE  "PID Statement Range Value = (PID_MAX - PID_MIN) For Use Elswhere" %
%   N24:20  PID_MIN  "PID Statement Minimum Value" %
%   N11:115  PT05_PID_MIN  "PT-05 Vacuum Transmitter No-5 PID Statement Minimum Input Value" %
%   N11:125  PT05_PID_MAX  "PT-05 Vacuum Transmitter No-5 PID Statement Maximum Input Value" %
%   N24:21  PID_MAX  "PID Statement Maximum Value" %
%   N11:105  PT05_PID_IN  "PT-05 Vacuum Transmitter No-5 PID Statement Input Value" %

